METHOD PROTECTED MS_SendingPosition2
VAR_INST
	lrPositionXFirstHalf  	: LREAL;
	lrPositionXSecondHalf  	: LREAL;
	lrPositionYFirstHalf  	: LREAL;
	lrPositionYSecondHalf 	: LREAL;
	lrRotationFirstHalf  	: LREAL;
	lrRotationSecondHalf	: LREAL;
END_VAR
CASE eCR800StateSendPosition OF 
	CR800_SEND_POSITION_CONVERTING:
		LTRUNC( lr_in := lrPositionX2,
				LTRUNC => lrPositionXFirstHalf);
		LTRUNC( lr_in := lrPositionY2,
				LTRUNC => lrPositionYFirstHalf);
		LTRUNC( lr_in := lrRotation2,
				LTRUNC => lrRotationFirstHalf);
	
		FRAC( lr_in := lrPositionX2,
				FRAC => lrPositionXSecondHalf);
		FRAC( lr_in := lrPositionY2,
				FRAC => lrPositionYSecondHalf);
		FRAC( lr_in := lrRotation2,
				FRAC => lrRotationSecondHalf);
				
		eCR800StateSendPosition := CR800_SEND_POSITION_SENDING;
		
	CR800_SEND_POSITION_SENDING:
		stCR800EthercatData.arrRegistersOutput[6028] :=	LREAL_TO_INT(lrPositionXFirstHalf); 
		stCR800EthercatData.arrRegistersOutput[6029] :=	LREAL_TO_INT(1000 * lrPositionXSecondHalf); 
		stCR800EthercatData.arrRegistersOutput[6030] :=	LREAL_TO_INT(lrPositionYFirstHalf); 
		stCR800EthercatData.arrRegistersOutput[6031] :=	LREAL_TO_INT(1000 * lrPositionYSecondHalf); 
		stCR800EthercatData.arrRegistersOutput[6032] :=	LREAL_TO_INT(lrRotationFirstHalf); 
		stCR800EthercatData.arrRegistersOutput[6033] :=	LREAL_TO_INT(1000 * lrRotationSecondHalf); 
			
		eCR800State := CR800_SEND_POSITION_2_DONE;
		
END_CASE
END_METHOD

METHOD PROTECTED MS_SendingPosition2Done
IF NOT bSendPosition2 THEN
	eCR800State := eCR800StateBeforeSendPosition;
	bBusy := FALSE;
	
END_IF
END_METHOD

METHOD Protected MS_Uninitialized
VAR_inst
	iLoop: INT;
END_VAR
//M_ResetVariables();

//M_OperationRigtsEnable(bRequest 	:= 0);
//eCR800StateDoRequest				:= 0 ;
eCR800StateHome 					:= 0 ;	
//eCR800StateReceiveCommand			:= 0 ;
//eCR800SendCommand					:= 0 ;
//eCR800StateInitializing 			:= 0 ;
eCR800StateCycleStop 				:= 0 ; 
eCR800StateCyclePause				:= 0 ; 
eCR800StateSendPosition				:= 0 ;

eErrorID := CR800_ERROR_OK;

bUninitialized := TRUE;
bInit := FALSE;
bGoHome := FALSE;
bUpdateRecipes := FALSE;
bGoAuto := FALSE;
bDoAction := FALSE;
bCycleStop := FALSE;
bCyclePause := FALSE;
bRestoreAuto := FALSE;
bRestoreCycle := FALSE;
bAbort := FALSE;
bError := FALSE;
bAutoModeStarted := FALSE;
bIsHomed := FALSE;
bReset := FALSE;
bStopped := FALSE;
bActive := FALSE; 
	
IF ServoIsOn THEN
	MR_Abort();
END_IF
END_METHOD

METHOD PROTECTED MS_UpdateRecipiesDone
IF NOT bUpdateRecipes THEN
	eCR800State := CR800_IDLE_HOMED ;
END_IF
END_METHOD

METHOD PROTECTED MS_UpdatingRecipies
IF M_DoRequest(iNumberOfRequest := E_RobotSystemActions.UPDATE_RECIPIES) THEN
	eCR800State := CR800_UPDATE_RECIPIES_DONE ;
END_IF
END_METHOD

PROPERTY Name : STRING
GET
Name := sName;
END_GET
SET
sName := Name;
END_SET
END_PROPERTY

(* Desription from CR800 side: Sets the validity of the operation rights for the
external signal control.. *)
{attribute 'monitoring' := 'variable'}
PROPERTY OperationRightsEnable : BOOL
GET
OperationRightsEnable := stCR800EthercatData.arrSignalsOutputConverted[6004] ;
END_GET
SET
stCR800EthercatData.arrSignalsOutputConverted[6004] := OperationRightsEnable ;
END_SET
END_PROPERTY

(*Desription from CR800 side:
Outputs the operation rights valid state for the
external signal control.
The operation right is given when the
operation right input signal is ON, the
controller mode is set to AUTOMATIC, and
there is no other device that currently has the
operation right.*)
{attribute 'monitoring' := 'variable'}
PROPERTY PUBLIC OperationRightsEnabled : BOOL
GET
OperationRightsEnabled := stCR800EthercatData.arrSignalsInputConverted[6004] ;
END_GET
END_PROPERTY

(* Reqest number that robot has to perform *)
{attribute 'monitoring' := 'variable'}
PROPERTY Override : USINT
GET
//Override :=	INT_TO_USINT(stCR800EthercatData.arrRegistersOutput[6021]);
Override := iOverride;
END_GET
SET
//stCR800EthercatData.arrRegistersOutput[6021] := USINT_TO_INT(iOverride);
iOverride := Override;
END_SET
END_PROPERTY

(* Desription from CR800 side:
"This output indicates that the program is
paused.
Turns ON when there is not slot multitask
running, and at least one slot is pausing.
However, slots whose starting condition is set
to ALWAYS or ERROR via a parameter
""SLT**"" will not be executed." *)
{attribute 'monitoring' := 'variable'}
PROPERTY PUBLIC Pausing : BOOL
GET
Pausing := stCR800EthercatData.arrSignalsInputConverted[6006] ;
END_GET
END_PROPERTY

(* Desription from CR800 side:
"This output indicates that a program is being
executed. During multitask operation, this
signal turns ON when at least one task slot is
operating.
However, slots whose starting condition is set
to ALWAYS or ERROR via a parameter ""SLT*""
will not be executed." *)
{attribute 'monitoring' := 'variable'}
PROPERTY PUBLIC ProgramOperating : BOOL
GET
ProgramOperating := stCR800EthercatData.arrSignalsInputConverted[6005] ;
END_GET
END_PROPERTY

(* Desription from CR800 side:
"This input cancels the paused status of the
program and brings the executing line to the
top. Executing a program reset makes it
possible to select a program.
In the multitask mode, the program reset is
applied to all task slots.
However, slots whose starting condition is set
to ALWAYS or ERROR via a parameter
""SLT**"" will not be executed." *)
{attribute 'monitoring' := 'variable'}
PROPERTY ProgramReset : BOOL
GET
ProgramReset := stCR800EthercatData.arrSignalsOutputConverted[6009] ;
END_GET
SET
stCR800EthercatData.arrSignalsOutputConverted[6009] := ProgramReset ;
END_SET
END_PROPERTY

(* "Outputs that in the program selection enabled
state.
Turns ON when program are not running or
pausing.
In multitask operation, this output turns ON
when all task slots are neither operating nor
paused.
However, slots whose starting condition is set
to ALWAYS or ERROR via a parameter
""SLT**"" will not be executed" *)
{attribute 'monitoring' := 'variable'}
PROPERTY PUBLIC ProgramSelectionEnabled : BOOL
GET
ProgramSelectionEnabled := stCR800EthercatData.arrSignalsInputConverted[6009] ;
END_GET
END_PROPERTY

(*Desription from CR800 side:
"This input starts a program. To start a specific
program, select the program using the
program selection signal ""PRGSEL"" and
numerical input ""IODATA,"" and then input the
start signal. Note that when the parameter
""PST"" is enabled, the system reads the
program number from the numerical input
(IODATA) and starts the corresponding
program (i.e., program selection becomes no
longer necessary).
All task slots are executed during multitask
operation.
However, slots whose starting condition is set
to ALWAYS or ERROR via a parameter ""SLT*""
will not be executed." *)
{attribute 'monitoring' := 'variable'}
PROPERTY ProgramStart : BOOL ;
GET
ProgramStart := stCR800EthercatData.arrSignalsOutputConverted[6005] ;
END_GET
SET
stCR800EthercatData.arrSignalsOutputConverted[6005] := ProgramStart ;
END_SET
END_PROPERTY

(* Desription from CR800 side:
This input stops the program being executed.
(The specification is the same as for the STOP
parameter.)
Unlike the STOP parameter, signal numbers
can be changed. *)
{attribute 'monitoring' := 'variable'}
PROPERTY ProgramStop2 : BOOL
GET
ProgramStop2 := stCR800EthercatData.arrSignalsOutputConverted[6007] ;
END_GET
SET
stCR800EthercatData.arrSignalsOutputConverted[6007] := ProgramStop2 ;
END_SET
END_PROPERTY

(* Desription from CR800 side:
"This output indicates that the program is
paused.
(The specification is the same as for the STOP
parameter.)" *)
{attribute 'monitoring' := 'variable'}
PROPERTY PUBLIC ProgramStopped : BOOL
GET
ProgramStopped := bStopped; // stCR800EthercatData.arrSignalsInputConverted[6007] ;
END_GET
END_PROPERTY

(* Reqest number that robot has to perform *)
{attribute 'monitoring' := 'variable'}
PROPERTY RequestNumber : UINT
GET
RequestNumber := iActionNumber;
END_GET
SET
stCR800EthercatData.arrRegistersOutput[6010] :=	UINT_TO_INT(RequestNumber);
END_SET
END_PROPERTY

PROPERTY SendingPosition1 : REFERENCE TO BOOL
GET
SendingPosition1 REF= bSendPosition1;
END_GET
END_PROPERTY

PROPERTY SendingPosition2 : REFERENCE TO BOOL
GET
SendingPosition2 REF= bSendPosition2;
END_GET
END_PROPERTY

(* Desription from a CR800 side:
"This input turns OFF the servo power supply
for the robot.(Applicable to all mechanisms)
The servo cannot be turned ON while this
signal is being input. *)
{attribute 'monitoring' := 'variable'}
PROPERTY PUBLIC ServoIsOff : BOOL
GET
ServoIsOff := NOT ServoIsOn AND CR800PoweredOn; //stCR800EthercatData.arrSignalsInputConverted[6012] ;
END_GET
END_PROPERTY

(* Desription from the CR800 side:
"This output turns ON when the servo power
supply for the robot is ON. If the servo power
supply is OFF, this output also remains OFF.
With a multi-mechanism configuration, this
output turns ON when the servo of at least one
mechanism is ON." *)
{attribute 'monitoring' := 'variable'}
PROPERTY PUBLIC ServoIsOn : BOOL
GET
ServoIsOn := stCR800EthercatData.arrSignalsInputConverted[6011] ;
END_GET
END_PROPERTY

(* Desription from a CR800 side:
"This input turns OFF the servo power supply
for the robot.(Applicable to all mechanisms)
The servo cannot be turned ON while this
signal is being input." *)
{attribute 'monitoring' := 'variable'}
PROPERTY ServoOFF : BOOL
GET
ServoOFF := stCR800EthercatData.arrSignalsOutputConverted[6012] ;
END_GET
SET
stCR800EthercatData.arrSignalsOutputConverted[6012] := ServoOFF ;
END_SET
END_PROPERTY

(* Descrition from the CR800 side:
"This input turns ON the servo power supply for
the robot.
With a multi-mechanism configuration, the
servo power supplies for all mechanisms will
be turned ON." *)
{attribute 'monitoring' := 'variable'}
PROPERTY ServoON : BOOL
GET
ServoON := stCR800EthercatData.arrSignalsOutputConverted[6011] ;
END_GET
SET
stCR800EthercatData.arrSignalsOutputConverted[6011] := ServoON ;
END_SET
END_PROPERTY

(* Actual state of main state machine *)
{attribute 'monitoring' := 'variable'}
PROPERTY State : REFERENCE TO E_CR800State
GET
State REF= eCR800State;
END_GET
END_PROPERTY

METHOD Protected StateMachine
VAR
	MS_CycleStopping_Done: INT;
END_VAR
CASE eCR800State OF
	CR800_UNINITIALIZED:
		MS_Uninitialized();
		
	CR800_INITIALIZING:
		MS_Initializing();
		
	CR800_READY_INITIALIZED:
		MS_ReadyInitialized();

	CR800_IDLE_NOT_HOMED:
		MS_IdleNotHomed();
		
	CR800_GOING_HOME:
		MS_GoingHome();
	
	CR800_GOING_HOME_DONE:
		MS_GoHomeDone();
		
	CR800_IDLE_HOMED:
		MS_IdleHomed();

	CR800_UPDATING_RECIPIES	:
		MS_UpdatingRecipies();
		
	CR800_UPDATE_RECIPIES_DONE:
		MS_UpdateRecipiesDone();
		
	CR800_GOING_AUTO:
		MS_GoingAuto();
		
	CR800_GOING_AUTO_DONE:
		MS_GoAutoDone();
		
	CR800_IDLE_AUTO:
		MS_IdleAuto();
		
	CR800_DOING_ACTION:
		MS_DoingAction();
		
	CR800_DOING_ACTION_DONE:
		MS_DoAction_Done();

	CR800_CYCLE_STOPPING:	
		MS_CycleStopping();
		
	CR800_CYCLE_STOPING_DONE:
		MS_CycleStopDone();
		
	CR800_IDLE_AUTO_PAUSED:
		MS_IdleAutoPaused();
		
	CR800_AUTO_RESTORING:
		MS_RestoringAuto();
	
	CR800_AUTO_RESTORING_DONE:
		MS_RestoreAutoDone();
		
	E_CR800State.CR800_CYCLE_PAUSING:
		MS_CyclePausing();
		
	E_CR800State.CR800_CYCLE_PAUSING_DONE:
		MS_CyclePauseDone();
	
	CR800_IDLE_CYCLE_PAUSED:
		MS_IdleCyclePaused();
	
	CR800_CYCLE_RESTORING:
		MS_RestoringCycle();
	
	CR800_CYCLE_RESTORING_DONE:
		MS_RestoreCycleDone();

	CR800_IN_EXTERNAL_ERROR:
		MS_InExternalError();
		
	CR800_SEND_POSITION_1:
		MS_SendingPosition1();
	
	CR800_SEND_POSITION_1_DONE:
		MS_SendingPosition1Done();	
		
	CR800_SEND_POSITION_2:
		MS_SendingPosition2();
	
	CR800_SEND_POSITION_2_DONE:
		MS_SendingPosition2Done();			
		
	CR800_RESET:
		MS_Reset();
		
	CR800_RESET_DONE:
		MS_ResetDone();
		
	CR800_ABORTING:
		MS_Aborting();
					
END_CASE
END_METHOD

(* Desription from CR800 side:
"Outputs that the stop is being input. (Logical
ADD of all devices.)" *)
{attribute 'monitoring' := 'variable'}
PROPERTY PUBLIC StopSTS : BOOL
GET
StopSTS := stCR800EthercatData.arrSignalsInputConverted[6008] ;
END_GET
END_PROPERTY

PROPERTY Uninitialized : REFERENCE TO BOOL
GET
Uninitialized REF= bUninitialized;
END_GET
END_PROPERTY

(*Desription from CR800 side:
This output indicates that the controller mode
is set to AUTOMATIC.*)
{attribute 'monitoring' := 'variable'}
{attribute 'monitoring' := 'call'}
PROPERTY  UserDefinedArea : ST_CR800UserDefinedArea
GET
UserDefinedArea.bArea1 := stCR800EthercatData.arrSignalsInputConverted[6241];
UserDefinedArea.bArea2 := stCR800EthercatData.arrSignalsInputConverted[6242];
UserDefinedArea.bArea3 := stCR800EthercatData.arrSignalsInputConverted[6243];
UserDefinedArea.bArea4 := stCR800EthercatData.arrSignalsInputConverted[6244];
UserDefinedArea.bArea5 := stCR800EthercatData.arrSignalsInputConverted[6245];
UserDefinedArea.bArea6 := stCR800EthercatData.arrSignalsInputConverted[6246];
UserDefinedArea.bArea7 := stCR800EthercatData.arrSignalsInputConverted[6247];
UserDefinedArea.bArea8 := stCR800EthercatData.arrSignalsInputConverted[6248];
END_GET
END_PROPERTY

PROPERTY UserDefinedArea1 : BOOL
GET
UserDefinedArea1 := stCR800EthercatData.arrSignalsInputConverted[6241];
END_GET
END_PROPERTY

PROPERTY UserDefinedArea2 : BOOL
GET
UserDefinedArea2 := stCR800EthercatData.arrSignalsInputConverted[6242];
END_GET
END_PROPERTY

PROPERTY UserDefinedArea3 : BOOL
GET
UserDefinedArea3 := stCR800EthercatData.arrSignalsInputConverted[6243];
END_GET
END_PROPERTY

PROPERTY UserDefinedArea4 : BOOL
GET
UserDefinedArea4 := stCR800EthercatData.arrSignalsInputConverted[6244];
END_GET
END_PROPERTY

PROPERTY UserDefinedArea5 : BOOL
GET
UserDefinedArea5 := stCR800EthercatData.arrSignalsInputConverted[6245];
END_GET
END_PROPERTY

PROPERTY UserDefinedArea6 : BOOL
GET
UserDefinedArea6 := stCR800EthercatData.arrSignalsInputConverted[6246];
END_GET
END_PROPERTY

PROPERTY UserDefinedArea7 : BOOL
GET
UserDefinedArea7 := stCR800EthercatData.arrSignalsInputConverted[6247];
END_GET
END_PROPERTY

PROPERTY UserDefinedArea8 : BOOL
GET
UserDefinedArea8 := stCR800EthercatData.arrSignalsInputConverted[6248];
END_GET
END_PROPERTY

END_FUNCTION_BLOCK

// ---- POUs/Machine/Module/RTCVision/FB_RTCVision.TcPOU
FUNCTION_BLOCK FB_RTCVision
VAR
	bFirstCycle			: BOOL := TRUE;	(* First cycle bit *)
	
	(* TCPIP params *)
	sName 				: STRING;		(* TCP/IP device name for other utilities *)
	sHost				: T_IPv4Addr;	(*  *)
	sAmsNetID 			: T_AmsNetID;	(*  *)
	iPort				: UINT;			(*  *)
	tTimeout			: TIME;			(*  *)
	
	(* Internal status *) 
	_bActive			: BOOL;			(* TCP/IP device initialized and ready to work *)
	_bBusy				: BOOL;			(* TCP/IP device is currently proccesing *)
	_bError				: BOOL;			(* Error occured while executing *)
	_iErrorID			: UDINT;		(* Error ID*)
	
	_bJobStarted		: BOOL;
	_bJobStopped		: BOOL;
	_eResult_Station1	: E_VisionResult;
	_eResult_Station2	: E_VisionResult;
	
	eCameraState		: E_RTCCameraState;		(* Current state of camera connection *)
	eCameraInitState	: E_RTCCameraInitState;		(* Current state of camera initialization *)
	eCameraMethodState	: E_RTCCameraMethodState;

	(* TCPIP communicate with Vision System - Service side is role as sever *)
	fbTcpClient 		: FB_TcpClient ;
	
	(* Messages buffers *)
	stSendData							: ST_TcpBufferData;		(*  *)
	stReciveData 						: ST_TcpBufferData;		(*  *)

	(* Temporary messeges *)
	sSendMessage 						: STRING;				(*  *)
	sReciveMessage						: STRING(1000);			(*  *)
	arrBufferMessage					: ARRAY[0..10] OF STRING;
	iMessageIndex	 					: INT;	
	sNewLine							: STRING := '$R$L';
	
	(* Rising edge trigger *)
	rtError								: R_TRIG; 					(* Rising edge trigger for function block error *)
	
	(* Status inormation and number *)
	iLastStatusCode						: INT; 
	sLastStatusCode						: STRING;

	(* Internal variables of methods *)
	eSetJobNumber							: E_VisionJob;
	eGetJobNumber							: E_VisionJob;
	eVisionResult							: E_VisionResult;
	
END_VAR

(* First cycle procedure *)
IF bFirstCycle THEN
	bFirstCycle := FALSE;
	
END_IF

_bActive := eCameraState >= RTC_CAMERA_READY;

(* Report errors that occur *)
rtError(CLK:=_bError);

IF rtError.Q THEN 
	fbMachineLogger.MR_AddLogs(FUN_MergeStrings5(sName, ' : Error occured (error ID: ', UDINT_TO_STRING(_iErrorID), ')', ''));

END_IF

(* Execute TCP/IP FB and timers *)
fbTcpClient();

(* Execute state machine *)
StateMachine();

PROPERTY Active  : REFERENCE TO BOOL
GET
Active REF= _bActive;
END_GET
END_PROPERTY

PROPERTY Busy : REFERENCE TO BOOL
GET
Busy REF= _bBusy;
END_GET
END_PROPERTY

PROPERTY CurrentJob : UINT
GET
END_GET
SET
END_SET
END_PROPERTY

PROPERTY Error : REFERENCE TO BOOL
GET
Error REF= _bError;
END_GET
END_PROPERTY

PROPERTY ErrorID : REFERENCE TO UDINT
GET
ErrorID REF= _iErrorID;
END_GET
END_PROPERTY

METHOD GetInfor : BOOL
VAR_INPUT
END_VAR
END_METHOD

PROPERTY JobStarted : BOOL
GET
END_GET
END_PROPERTY

PROPERTY JobStopped : BOOL
GET
END_GET
END_PROPERTY

METHOD MR_Abort : BOOL
VAR_INPUT
END_VAR
IF eCameraState >= RTC_CAMERA_READY THEN
	_bBusy := TRUE;
	MR_Abort := FALSE;
	eCameraState := RTC_CAMERA_ABORTING;
	fbMachineLogger.MR_AddLogs(CONCAT(sName,' : abort requested'));	
	
ELSIF eCameraState = RTC_CAMERA_UNINITIALIZED THEN
	_bBusy := FALSE;
	MR_Abort := TRUE;
	fbMachineLogger.MR_AddLogs(CONCAT(sName,' : abort done'));	
	
END_IF
END_METHOD

METHOD MR_Clear : BOOL
VAR_INPUT
END_VAR
IF eCameraState = RTC_CAMERA_IDLE THEN
	_bBusy := TRUE;
	MR_Clear := FALSE;
	eCameraState := RTC_CAMERA_CLEAR_DATA;
	fbMachineLogger.MR_AddLogs(CONCAT(sName,' : Clear data requested'));	
	
ELSIF eCameraState = RTC_CAMERA_METHOD_DONE THEN
	_bBusy := FALSE;
	MR_Clear := TRUE;
	fbMachineLogger.MR_AddLogs(CONCAT(sName,' : Clear data done'));	

END_IF
END_METHOD

METHOD MR_FirstCycle : BOOL
VAR_INPUT
	sCameraName 			: STRING;		(*  *)
	sClientHost				: T_IPv4Addr;	(*  *)
	sClientAmsNetID 		: T_AmsNetID;	(*  *)
	iClientPort				: UINT;			(*  *)
	tTimeout				: TIME;			(*  *)
	
END_VAR
(* Set fixture name *)
THIS^.sName := sCameraName;

(* Set fixture server initial parameters *)
THIS^.fbTcpClient.MR_FirstCycle(	sName 		:= CONCAT('TCP/IP client of ',sCameraName),
									sHost		:= sClientHost,
									sAmsNetID	:= sClientAmsNetID,
									iPort 		:= iClientPort,
									tTimeout 	:= tTimeout);
END_METHOD

METHOD MR_GetBatchInfor : BOOL
VAR_INPUT
END_VAR
IF eCameraState = RTC_CAMERA_IDLE THEN	
	_bBusy := TRUE;
	MR_GetBatchInfor := FALSE;
	eCameraState := RTC_CAMERA_GET_BATCH_DATA;
	fbMachineLogger.MR_AddLogs(CONCAT(sName,' : get batch data requested'));
	
ELSIF eCameraState = RTC_CAMERA_METHOD_DONE THEN
	_bBusy := FALSE;
	MR_GetBatchInfor := TRUE;
	fbMachineLogger.MR_AddLogs(CONCAT(sName,' : get batch data done'));

END_IF
END_METHOD

METHOD MR_GetResult : BOOL
VAR_INPUT
END_VAR
IF eCameraState = RTC_CAMERA_IDLE THEN	
	_bBusy := TRUE;
	MR_GetResult := FALSE;
	eCameraState := RTC_CAMERA_GET_RESULT;
	fbMachineLogger.MR_AddLogs(CONCAT(sName,' : get result requested'));
	
ELSIF eCameraState = RTC_CAMERA_METHOD_DONE THEN
	_bBusy := FALSE;
	MR_GetResult := TRUE;
	fbMachineLogger.MR_AddLogs(CONCAT(sName,' : get result done'));

END_IF
END_METHOD

METHOD MR_Init : BOOL
VAR_INPUT
END_VAR
IF eCameraState = RTC_CAMERA_UNINITIALIZED THEN
	_bBusy := TRUE;
	MR_Init := FALSE;
	eCameraState := RTC_CAMERA_INITIALIZING;
	fbMachineLogger.MR_AddLogs(CONCAT(sName,' : initializing requested'));	

ELSIF eCameraState >= RTC_CAMERA_READY THEN
	_bBusy := FALSE;
	MR_Init := TRUE;
	fbMachineLogger.MR_AddLogs(CONCAT(sName,' : initializing done'));
	
END_IF
END_METHOD

METHOD MR_Reset : BOOL
VAR_INPUT
END_VAR
END_METHOD

METHOD MR_SetJob : BOOL
VAR_INPUT
	eSetJobNumber 		: E_VisionJob;
END_VAR
IF eCameraState = RTC_CAMERA_IDLE THEN
	THIS^.eSetJobNumber := eSetJobNumber;
	_bBusy := TRUE;
	MR_SetJob := FALSE;
	eCameraState := RTC_CAMERA_SET_JOB;
	fbMachineLogger.MR_AddLogs(FUN_MergeStrings4(sName,' : setting job ',TO_STRING(eSetJobNumber),' requested'));
	
ELSIF eCameraState = RTC_CAMERA_METHOD_DONE THEN
	_bBusy := FALSE;
	MR_SetJob := TRUE;
	fbMachineLogger.MR_AddLogs(FUN_MergeStrings4(sName,' : setting job ',TO_STRING(eSetJobNumber),' done'));

END_IF
END_METHOD

METHOD MR_Start : BOOL
VAR_INPUT
END_VAR
IF eCameraState = RTC_CAMERA_IDLE THEN
	_bBusy := TRUE;
	MR_Start := FALSE;
	eCameraState := RTC_CAMERA_START;
	fbMachineLogger.MR_AddLogs(CONCAT(sName,' : Start job requested'));	
	
ELSIF eCameraState = RTC_CAMERA_METHOD_DONE THEN
	_bBusy := FALSE;
	MR_Start := TRUE;
	fbMachineLogger.MR_AddLogs(CONCAT(sName,' : Start job done'));	

END_IF
END_METHOD

METHOD MR_Stop : BOOL
VAR_INPUT
END_VAR
IF eCameraState = RTC_CAMERA_IDLE THEN	
	_bBusy := TRUE;
	MR_Stop := FALSE;
	eCameraState := RTC_CAMERA_STOP;
	fbMachineLogger.MR_AddLogs(CONCAT(sName,' : stop job requested'));
	
ELSIF eCameraState = RTC_CAMERA_METHOD_DONE THEN
	_bBusy := FALSE;
	MR_Stop := TRUE;
	fbMachineLogger.MR_AddLogs(CONCAT(sName,' : stop job done'));

END_IF
END_METHOD

METHOD MR_StopCycle : BOOL
VAR_INPUT
END_VAR
IF eCameraState = RTC_CAMERA_IDLE THEN	
	_bBusy := TRUE;
	MR_StopCycle := FALSE;
	eCameraState := RTC_CAMERA_STOP_CYCLE;
	fbMachineLogger.MR_AddLogs(CONCAT(sName,' : stop current cycle requested'));
	
ELSIF eCameraState = RTC_CAMERA_METHOD_DONE THEN
	_bBusy := FALSE;
	MR_StopCycle := TRUE;
	fbMachineLogger.MR_AddLogs(CONCAT(sName,' : stop current cycle done'));

END_IF
END_METHOD

METHOD PROTECTED MS_Aborting
fbTcpClient.MR_Abort();

IF NOT fbTcpClient.Active THEN 
	//IF M_ResetParameters() THEN
		eCameraState := RTC_CAMERA_UNINITIALIZED;
		
	//END_IF	
END_IF
END_METHOD

METHOD PROTECTED MS_GetJob : BOOL
VAR_INPUT
END_VAR
CASE eCameraMethodState OF
	RTC_CAMERA_METHOD_SEND_COMMAND:
		MEMSET(ADR(sSendMessage),0,SIZEOF(sSendMessage));
		sSendMessage := CONCAT('GJ','$R$L');
		FUN_StringToTcpBufferData(ADR(sSendMessage),ADR(stSendData));
		
		IF fbTcpClient.MR_AppendToSendBuffer(stSendData) THEN
			eCameraMethodState := RTC_CAMERA_METHOD_RECEIVE_RESPONSE;

		END_IF
		
	RTC_CAMERA_METHOD_RECEIVE_RESPONSE:
		stReciveData := fbTcpClient.NextRecivedMessage;
		
		IF stReciveData.iLength > 0 THEN
			MEMSET(ADR(sReciveMessage),0,SIZEOF(sReciveMessage));
			FUN_TcpBufferDataToString(ADR(sReciveMessage),ADR(stReciveData));

			IF sReciveMessage = 'GJ1' THEN
				THIS^.eGetJobNumber := CASE_RECEIVER_E25_0100812762;				
			END_IF
			
			eCameraMethodState := RTC_CAMERA_METHOD_SEND_COMMAND;
			eCameraState := RTC_CAMERA_METHOD_DONE;	
		END_IF
		
END_CASE
END_METHOD

METHOD PROTECTED MS_Idle
;
END_METHOD

METHOD PROTECTED MS_Initializing
CASE eCameraInitState OF
	
	RTC_INIT_CONNECTION:
		fbTcpClient.MR_Init();
		
		IF fbTcpClient.Active THEN
			eCameraInitState := RTC_INIT_CLEAR_BUFFER;
			
		ELSIF fbTcpClient.Error THEN
			_bError := TRUE;
			_iErrorID := fbTcpClient.ErrorID;
			
		END_IF
	
	RTC_INIT_CLEAR_BUFFER:
		fbTcpClient.MR_ClearAllBuffers();
		eCameraInitState := RTC_INIT_WAIT_FOR_CONFIRMATION;
		
		IF fbTcpClient.Error THEN
			_bError := TRUE;
			_iErrorID := fbTcpClient.ErrorID;
			
		END_IF

	RTC_INIT_WAIT_FOR_CONFIRMATION:
		stReciveData := fbTcpClient.NextRecivedMessage;

		IF stReciveData.iLength > 0 THEN
			MEMSET(ADR(sReciveMessage),0,SIZEOF(sReciveMessage));
			FUN_TcpBufferDataToString(ADR(sReciveMessage),ADR(stReciveData));
	
			IF sReciveMessage = 'User Logged In' THEN
				eCameraInitState := RTC_INIT_DONE;
			
			END_IF
		ELSIF fbTcpClient.Error THEN
			_bError := TRUE;
			_iErrorID := fbTcpClient.ErrorID;
			
		END_IF
		
	RTC_INIT_DONE:
		eCameraInitState := RTC_INIT_CONNECTION;
		eCameraState := RTC_CAMERA_READY;
END_CASE
END_METHOD

METHOD PROTECTED MS_MethodDone
IF NOT _bBusy THEN
	eCameraState := RTC_CAMERA_IDLE;
	
END_IF
END_METHOD

METHOD PROTECTED MS_Ready
eCameraState := RTC_CAMERA_IDLE;
END_METHOD

METHOD PROTECTED MS_Result
CASE eCameraMethodState OF
	RTC_CAMERA_METHOD_SEND_COMMAND:
		MEMSET(ADR(sSendMessage),0,SIZEOF(sSendMessage));
		sSendMessage := CONCAT('Result','$R$L');
		FUN_StringToTcpBufferData(ADR(sSendMessage),ADR(stSendData));
		
		IF fbTcpClient.MR_AppendToSendBuffer(stSendData) THEN
			eCameraMethodState := RTC_CAMERA_METHOD_RECEIVE_RESPONSE;

		END_IF
		
	RTC_CAMERA_METHOD_RECEIVE_RESPONSE:
		stReciveData := fbTcpClient.NextRecivedMessage;
		
		IF stReciveData.iLength > 0 THEN
			MEMSET(ADR(sReciveMessage),0,SIZEOF(sReciveMessage));
			FUN_TcpBufferDataToString(ADR(sReciveMessage),ADR(stReciveData));
			
			IF sReciveMessage = 'ResultGood' THEN
				eVisionResult := VISION_RESULT_GOOD;
				
			ELSIF sReciveMessage = 'ResultDirt' THEN
				eVisionResult := VISION_RESULT_CONTAMINATION_DIRTY;
				
			ELSIF sReciveMessage = 'ResultDent' THEN
				eVisionResult := VISION_RESULT_SCRATCH_DENT;
				
			ELSIF sReciveMessage = 'ResultReject' THEN
				eVisionResult := VISION_RESULT_REJECT;
				
			ELSE
				eVisionResult := VISION_RESULT_UNKNOWN;
				
			END_IF			
			eCameraMethodState := RTC_CAMERA_METHOD_SEND_COMMAND;
			eCameraState := RTC_CAMERA_METHOD_DONE;	
			
		END_IF		
END_CASE
END_METHOD

METHOD PROTECTED MS_SetJob
CASE eCameraMethodState OF
	RTC_CAMERA_METHOD_SEND_COMMAND:
		MEMSET(ADR(sSendMessage),0,SIZEOF(sSendMessage));
		sSendMessage := FUN_MergeStrings3('SJ', TO_STRING(TO_INT(THIS^.eSetJobNumber)), '$R$L');
		FUN_StringToTcpBufferData(ADR(sSendMessage),ADR(stSendData));
		
		IF fbTcpClient.MR_AppendToSendBuffer(stSendData) THEN
			eCameraMethodState := RTC_CAMERA_METHOD_RECEIVE_RESPONSE;

		END_IF
		
	RTC_CAMERA_METHOD_RECEIVE_RESPONSE:
		stReciveData := fbTcpClient.NextRecivedMessage;
		
		IF stReciveData.iLength > 0 THEN
			MEMSET(ADR(sReciveMessage),0,SIZEOF(sReciveMessage));
			FUN_TcpBufferDataToString(ADR(sReciveMessage),ADR(stReciveData));
			
			IF sReciveMessage = 'SJDone' THEN
				eCameraMethodState := RTC_CAMERA_METHOD_SEND_COMMAND;
				eCameraState := RTC_CAMERA_METHOD_DONE;			
			END_IF	
		END_IF
		
END_CASE
END_METHOD

METHOD PROTECTED MS_Start
CASE eCameraMethodState OF
	
	RTC_CAMERA_METHOD_SEND_COMMAND:
		MEMSET(ADR(sSendMessage),0,SIZEOF(sSendMessage));
		sSendMessage := CONCAT('Start', '$R$L');
		FUN_StringToTcpBufferData(ADR(sSendMessage),ADR(stSendData));
		
		IF fbTcpClient.MR_AppendToSendBuffer(stSendData) THEN
			eCameraMethodState := RTC_CAMERA_METHOD_RECEIVE_RESPONSE;
							
		END_IF
		
	RTC_CAMERA_METHOD_RECEIVE_RESPONSE:
		stReciveData := fbTcpClient.NextRecivedMessage;
		
		IF stReciveData.iLength > 0 THEN
			MEMSET(ADR(sReciveMessage),0,SIZEOF(sReciveMessage));
			FUN_TcpBufferDataToString(ADR(sReciveMessage),ADR(stReciveData));
			
			IF sReciveMessage = 'StartDone' THEN
				eCameraMethodState := RTC_CAMERA_METHOD_SEND_COMMAND;
				eCameraState := RTC_CAMERA_METHOD_DONE;			
			END_IF	
		END_IF

END_CASE
END_METHOD

METHOD PROTECTED MS_Stop : BOOL
VAR_INPUT
END_VAR
CASE eCameraMethodState OF
	RTC_CAMERA_METHOD_SEND_COMMAND:
		MEMSET(ADR(sSendMessage),0,SIZEOF(sSendMessage));
		sSendMessage := CONCAT('Stop','$R$L');
		FUN_StringToTcpBufferData(ADR(sSendMessage),ADR(stSendData));
		
		IF fbTcpClient.MR_AppendToSendBuffer(stSendData) THEN
			eCameraMethodState := RTC_CAMERA_METHOD_RECEIVE_RESPONSE;

		END_IF
		
	RTC_CAMERA_METHOD_RECEIVE_RESPONSE:
		stReciveData := fbTcpClient.NextRecivedMessage;
		
		IF stReciveData.iLength > 0 THEN
			MEMSET(ADR(sReciveMessage),0,SIZEOF(sReciveMessage));
			FUN_TcpBufferDataToString(ADR(sReciveMessage),ADR(stReciveData));
			
			IF sReciveMessage = 'StopDone' THEN
				eCameraMethodState := RTC_CAMERA_METHOD_SEND_COMMAND;
				eCameraState := RTC_CAMERA_METHOD_DONE;			
			END_IF	
		END_IF
		
END_CASE
END_METHOD

METHOD PROTECTED MS_Uninitialized
;
END_METHOD

METHOD PROTECTED StateMachine : BOOL
VAR_INPUT
END_VAR
CASE eCameraState OF
	RTC_CAMERA_UNINITIALIZED:
		MS_Uninitialized();
	
	RTC_CAMERA_INITIALIZING:
		MS_Initializing();
		
	RTC_CAMERA_READY:
		MS_Ready();
		
	RTC_CAMERA_IDLE:
		MS_Idle();
		
	RTC_CAMERA_SET_JOB:
		MS_SetJob();
		

	
	RTC_CAMERA_METHOD_DONE:
		MS_MethodDone();
		
	RTC_CAMERA_ABORTING:
		MS_Aborting();
END_CASE
END_METHOD

END_FUNCTION_BLOCK

// ---- POUs/Libs/Bowl Feeder/FB_BowlFeeder.TcPOU
(*
Copyrights	: Operation Automation Department
Author		: HVAP
Description	: This function block is used to control bowl feeder REOVIB MFS 268
*)
FUNCTION_BLOCK FB_BowlFeeder IMPLEMENTS I_BowlFeeder
VAR CONSTANT
	(* STRINGS *)
	sPRODUCT_PRESENCE_SENSOR_NAME	: STRING := 'Producr presence sensor';
	sSTATUS_RELAY					: STRING := 'Status relay from bowl driver';
	sENABLE							: STRING := 'Enable bowl driver';
END_VAR
VAR
	bFirstCycle			: BOOL := TRUE;		(* First cycle bit *)
	sName 				: STRING;			(* Bowl Feeder name for other utilities *)	
	
	(* Internal status *)
	_bActive : BOOL;
	_bBusy : BOOL;
	_bError : BOOL;
	_uiErrorID : UINT;
	
	(* State machine *)
	eBowlFeederUnitState 		: E_BowlFeederUnitState;
	eBowlFeederUnitStateInit 	: E_BowlFeederUnitStateInit;
	
	(* Hardware module *)
	//_diProductPresence	: FB_DigitalInput;	(* Sensor for monitoring the queue of components on the track or an input for switching to the second setpoint 24 VDC (PNP). *)
	diStatusRelay		: FB_DigitalInput;	(* Relay closes when the feeder is running – the relay opens when there is no enable signal or a fault displayed. *)
	doEnable			: FB_DigitalOutput;	(* External control function to switch the power output ON or OFF *)
	_aoSetpoint			: FB_AnalogOutput;	(* 0-100%*)
	
	(* Rising edge trigger *)
	rtError								: R_TRIG; 					(* Rising edge trigger for function block error *)
END_VAR
(*
Version history:

+-------------+------------+----------------+----------+------------------------------------------+
|Date         | Version    | created under  | Author   | Remark                                   |
+=============+============+================+==========+==========================================+
|2024-02      | 1.0.0.0    | V3.1.4024.22   | HVAP     | Function block created                   |
+-------------+------------+----------------+----------+------------------------------------------+

*)

IF bFirstCycle THEN
	bFirstCycle := FALSE;
	
//	_diProductPresence.MR_FirstCycle( 	sName 		:= CONCAT(STR1:= sName, STR2:= CONCAT(STR1:= ':', STR2:= sPRODUCT_PRESENCE_SENSOR_NAME)),
//										sModuleType := '',
//										sPortID 	:= '');
	
	diStatusRelay.MR_FirstCycle(	sName		:= CONCAT(STR1:= sName, STR2:= CONCAT(STR1:= ':', STR2:= sSTATUS_RELAY)),
									sModuleType	:= '',
									sPortID		:= '');
									
	doEnable.MR_FirstCycle(	sName		:= CONCAT(STR1:= sName, STR2:= CONCAT(STR1:= ':', STR2:= sENABLE)),
							sModuleType	:= '',
							sPortID		:= '');
END_IF

(* Ready to work *)
_bActive := eBowlFeederUnitState >= BOWL_FEEDER_UNIT_IDLE;
_bBusy := eBowlFeederUnitState <> BOWL_FEEDER_UNIT_IDLE AND eBowlFeederUnitState <> BOWL_FEEDER_UNIT_UNINITIALIZED;

(* Report errors that occur *)
rtError(CLK:=_bError);
IF rtError.Q THEN 
	fbMachineLogger.MR_AddLogs(CONCAT(sName, ' : Error occured'));
END_IF

StateMachine();

PROPERTY Active : BOOL
GET
Active := _bActive;
END_GET
END_PROPERTY

PROPERTY Busy : BOOL
GET
Busy := _bBusy;
END_GET
END_PROPERTY

PROPERTY Error : BOOL
GET
Error := _bError;
END_GET
END_PROPERTY

PROPERTY ErrorID : UINT
GET
ErrorID := _uiErrorID;
END_GET
END_PROPERTY

METHOD MR_FirstCycle : BOOL
VAR_INPUT
	sName	: STRING;
END_VAR
THIS^.sName := sName;
END_METHOD

METHOD MR_Init : BOOL
VAR_INPUT
END_VAR
IF eBowlFeederUnitState = BOWL_FEEDER_UNIT_UNINITIALIZED THEN
	MR_Init := FALSE;
	eBowlFeederUnitState := BOWL_FEEDER_UNIT_INITIALIZING;	
	fbMachineLogger.MR_AddLogs(CONCAT(sName,': initializing requested'));
		
ELSIF eBowlFeederUnitState >= BOWL_FEEDER_UNIT_READY_INITIALIZED THEN
	MR_Init := TRUE;
	fbMachineLogger.MR_AddLogs(CONCAT(sName,': initializing done'));

END_IF
END_METHOD

METHOD MR_Start : BOOL
VAR_INPUT
END_VAR
IF eBowlFeederUnitState = BOWL_FEEDER_UNIT_IDLE THEN
	MR_Start := FALSE;
	eBowlFeederUnitState := BOWL_FEEDER_UNIT_START;
	fbMachineLogger.MR_AddLogs(CONCAT(sName,': Start requesting'));
		
ELSIF eBowlFeederUnitState = BOWL_FEEDER_UNIT_RUNNING THEN
	MR_Start := TRUE;
	fbMachineLogger.MR_AddLogs(CONCAT(sName,': Start done, is running'));
	
END_IF
END_METHOD

METHOD MR_Stop : BOOL
VAR_INPUT
END_VAR
IF eBowlFeederUnitState = BOWL_FEEDER_UNIT_IDLE THEN
	MR_Stop := FALSE;
	eBowlFeederUnitState := BOWL_FEEDER_UNIT_STOP;
	fbMachineLogger.MR_AddLogs(CONCAT(sName,': Stop requesting'));

ELSIF eBowlFeederUnitState = BOWL_FEEDER_UNIT_IDLE THEN
	MR_Stop := TRUE;
	fbMachineLogger.MR_AddLogs(CONCAT(sName,': Stop done'));
	
END_IF
END_METHOD

METHOD MS_Abort
doEnable.Out := FALSE;

IF NOT diStatusRelay.In THEN
	(* Status bit *)
	_bError		:= FALSE;
	
	(* State transition *)
	eBowlFeederUnitState := BOWL_FEEDER_UNIT_UNINITIALIZED;
END_IF
END_METHOD

METHOD PROTECTED MS_Idle
;
END_METHOD

METHOD PROTECTED MS_Initializing
CASE eBowlFeederUnitStateInit OF
	BOWL_FEEDER_UNIT_INIT_START:
		doEnable.Out := TRUE;
		eBowlFeederUnitStateInit := BOWL_FEEDER_UNIT_INIT_RUNNING_CHECK;
		
	BOWL_FEEDER_UNIT_INIT_RUNNING_CHECK:
		IF diStatusRelay.In THEN
			eBowlFeederUnitStateInit := BOWL_FEEDER_UNIT_INIT_STOP;
		END_IF
	
	BOWL_FEEDER_UNIT_INIT_STOP:
		doEnable.Out := FALSE;
		eBowlFeederUnitStateInit := BOWL_FEEDER_UNIT_INIT_STOP_CHECK;
		
	BOWL_FEEDER_UNIT_INIT_STOP_CHECK:
		IF NOT diStatusRelay.In THEN
			eBowlFeederUnitStateInit := BOWL_FEEDER_UNIT_INIT_DONE;
		END_IF
		
	BOWL_FEEDER_UNIT_INIT_DONE:
		eBowlFeederUnitStateInit := BOWL_FEEDER_UNIT_INIT_START;
		eBowlFeederUnitState := BOWL_FEEDER_UNIT_READY_INITIALIZED;
		
END_CASE
END_METHOD

METHOD PROTECTED MS_Ready
eBowlFeederUnitState := BOWL_FEEDER_UNIT_IDLE;
END_METHOD

METHOD MS_Running
eBowlFeederUnitState := BOWL_FEEDER_UNIT_IDLE;
END_METHOD

METHOD PROTECTED MS_Start : BOOL
VAR_INPUT
END_VAR
doEnable.Out := TRUE;

IF diStatusRelay.In THEN
	eBowlFeederUnitState := BOWL_FEEDER_UNIT_RUNNING;
END_IF
END_METHOD

METHOD MS_Stop
doEnable.Out := FALSE;

IF NOT diStatusRelay.In THEN
	eBowlFeederUnitState := BOWL_FEEDER_UNIT_STOP_DONE;
END_IF
END_METHOD

METHOD MS_StopDone
eBowlFeederUnitState := BOWL_FEEDER_UNIT_IDLE;
END_METHOD

METHOD PROTECTED MS_Uninitialized
;
END_METHOD

PROPERTY Running : BOOL
GET
Running := diStatusRelay.In;
END_GET
END_PROPERTY

PROPERTY Setpoint : REAL
GET
Setpoint := _aoSetpoint.Value;
END_GET
SET
_aoSetpoint.Value := Setpoint;
END_SET
END_PROPERTY

METHOD PROTECTED StateMachine
CASE eBowlFeederUnitState OF
	BOWL_FEEDER_UNIT_UNINITIALIZED:
		MS_Uninitialized();
		
	BOWL_FEEDER_UNIT_INITIALIZING:
		MS_Initializing();
		
	BOWL_FEEDER_UNIT_READY_INITIALIZED:
		MS_Ready();
		
	BOWL_FEEDER_UNIT_IDLE:
		MS_Idle();
		
	BOWL_FEEDER_UNIT_START:
		MS_Start();
		
	BOWL_FEEDER_UNIT_RUNNING:
		MS_Running();
		
	BOWL_FEEDER_UNIT_STOP:
		MS_Stop();
		
	BOWL_FEEDER_UNIT_STOP_DONE:
		MS_StopDone();
		
	BOWL_FEEDER_UNIT_ABORT:
		MS_Abort();
	
END_CASE
END_METHOD

END_FUNCTION_BLOCK

// ---- POUs/Libs/Analog Devices/Analog Output/FB_AnalogOutput.TcPOU
(* 
| :Description: This function block represents basic analog output and can be used for creating an instance of analog output device. 
| To control the output state use property "Out" 
*)
FUNCTION_BLOCK FB_AnalogOutput EXTENDS FB_AnalogDevice IMPLEMENTS I_AnalogOutput
VAR
	intAnalogOut AT %Q* : INT; (* Analog output value 0-32767 *)
	rConvertedValue : REAL;
END_VAR
(*
Version history:

+-------------+------------+----------------+----------+------------------------------------------+
|Date         | Version    | created under  | Author   | Remark                                   |
+=============+============+================+==========+==========================================+
|2024-02      | 1.0.0.0    | V3.1.4024.22   | HVAP     | Function block created                   |
+-------------+------------+----------------+----------+------------------------------------------+

*)

(*
Analog output
0-10V : 0-32767 : 0-100%
*)

PROPERTY Value : REAL
GET
Value := (INT_TO_REAL(intAnalogOut)/32767.0)*100.0;
END_GET
SET
intAnalogOut := REAL_TO_INT((Value/(100.0 - 0.0))*(32767.0 - 0.0));
END_SET
END_PROPERTY

END_FUNCTION_BLOCK

// ---- POUs/Libs/Analog Devices/Analog Device/FB_AnalogDevice.TcPOU
(* 
:Description: This function block is base for all other analog devices.
*)
FUNCTION_BLOCK ABSTRACT FB_AnalogDevice IMPLEMENTS I_AnalogDevice
VAR
	sName 		: STRING; (* Name of analog device instance *)
	sModuleType : STRING; (* Name of analog device instance *)
	sPortID		: STRING; (* Slot number on the module *)
END_VAR
(*
Version history:

+-------------+------------+----------------+----------+------------------------------------------+
|Date         | Version    | created under  | Author   | Remark                                   |
+=============+============+================+==========+==========================================+
|2024-02      | 1.0.0.0    | V3.1.4024.22   | HVAP     | Function block created                   |
+-------------+------------+----------------+----------+------------------------------------------+

*)

PROPERTY ModuleType : REFERENCE TO STRING
GET
ModuleType REF= sModuleType;
END_GET
END_PROPERTY

(*
:Description: Call this method in the first cycle of the program
*)
METHOD MR_FirstCycle : BOOL
VAR_INPUT
	sName		: STRING;
	sModuleType	: STRING;
	sPortID		: STRING;
END_VAR
THIS^.sName 		:= sName;
THIS^.sModuleType 	:= sModuleType;
THIS^.sPortID 		:= sPortID;
END_METHOD

PROPERTY Name : REFERENCE TO STRING
GET
Name REF= sName;
END_GET
END_PROPERTY

PROPERTY PortID : REFERENCE TO STRING
GET
PortID REF= sPortID;
END_GET
END_PROPERTY

END_FUNCTION_BLOCK

// ---- POUs/Machine/Module/RTCVision/FB_DoubleTrigger.TcPOU
FUNCTION_BLOCK FB_DoubleTrigger
VAR
	doCam : FB_DigitalOutput;
END_VAR

METHOD Command : BOOL
VAR_INPUT	
	PulseWidth	: TIME; //T#0.1ms
	DelayTimeForSecondTrigger	: TIME; //T#0.1ms
END_VAR
VAR_INST
	uiState 					: UINT;
	tonDelay					: TON;
END_VAR
CASE uiState OF
	0://first trigger on
		doCam.Out := TRUE;
		uiState := 10;
	10://first trigger off
		tonDelay(IN := TRUE, PT := PulseWidth);
		IF tonDelay.Q THEN	
			doCam.Out := FALSE;	
			tonDelay(IN := FALSE);
			uiState := 20;
		END_IF
	20://second trigger on
		tonDelay(IN := TRUE, PT := DelayTimeForSecondTrigger);
		IF tonDelay.Q THEN	
			doCam.Out := TRUE;
			tonDelay(IN := FALSE);
			uiState := 30;
		END_IF
	30://second trigger off
		tonDelay(IN := TRUE, PT := PulseWidth); 
		IF tonDelay.Q THEN
			doCam.Out := FALSE;
			tonDelay(IN := FALSE);
			Command := TRUE;
			uiState := 0;
		END_IF
END_CASE
END_METHOD

END_FUNCTION_BLOCK

// ---- POUs/Libs/Utilities/FB_DataSetFifo_1.TcPOU
FUNCTION_BLOCK FB_DataSetFifo_1
VAR_INPUT
	bOverwrite	: BOOL;
	in 			: LREAL;
END_VAR
VAR_OUTPUT
	bOk			: BOOL;
	nCount		: UDINT;
	nLoad		: UDINT;
	out			: LREAL;
END_VAR
VAR
	arrBuffer 	: ARRAY[0..10000] OF BYTE; (* Buffer memory used by FB_MemRingBuffer function block *)
	fbBuffer	: FB_MemRingBuffer;
END_VAR

;

ACTION A_Add:
fbBuffer.A_AddTail( pWrite:= ADR( in ),
					cbWrite:= SIZEOF( in ),
					pBuffer:= ADR( arrBuffer ),
					cbBuffer:= SIZEOF( arrBuffer ),
					bOk=> bOk,
					nCount => nCount );


IF NOT bOk THEN (* overflow ? *)
	IF bOverwrite THEN
		fbBuffer.A_RemoveHead(); (* remove one oldest entry *)

		fbBuffer.A_AddTail( bOk => bOk, nCount => nCount );
	END_IF
END_IF



nLoad := (fbBuffer.cbSize * 100) / 10000;
END_ACTION

ACTION A_Get:
fbBuffer.A_GetHead( pRead:= ADR( out ),
					cbRead:= SIZEOF( out ),
					pBuffer:= ADR( arrBuffer ),
					cbBuffer:= SIZEOF( arrBuffer ),
					bOk=> bOk,
					nCount => nCount );

nLoad := (fbBuffer.cbSize * 100) / 10000;
END_ACTION

ACTION A_Remove:
fbBuffer.A_RemoveHead( 	pRead:= ADR( out ),
						cbRead:= SIZEOF( out ),
						pBuffer:= ADR( arrBuffer ),
						cbBuffer:= SIZEOF( arrBuffer ),
						bOk=> bOk,
						nCount => nCount );

nLoad := (fbBuffer.cbSize * 100) / 10000;
END_ACTION

ACTION A_Reset:
MEMSET( ADR( arrBuffer ), 0, SIZEOF( arrBuffer ) ); (* reset (optional) internal buffer *)

fbBuffer.A_Reset( 	bOk=> bOk,
					nCount => nCount );

nLoad := (fbBuffer.cbSize * 100) / 10000;
END_ACTION

END_FUNCTION_BLOCK

// ---- POUs/Libs/Utilities/FB_DataSetFifo.TcPOU
FUNCTION_BLOCK FB_DataSetFifo
VAR
	arrBuffer 	: ARRAY[0..10000] OF BYTE; (* Buffer memory used by FB_MemRingBuffer function block *)
	fbBuffer	: FB_MemRingBuffer;
	
	_bOk		: BOOL;
	_nCount		: UDINT;
	_nLoad		: UDINT;
	_bOverwrite	: BOOL;
END_VAR

METHOD Add1Data : BOOL
VAR_INPUT
	in : LREAL;
END_VAR
fbBuffer.A_AddTail( pWrite:= ADR( in ),
					cbWrite:= SIZEOF( in ),
					pBuffer:= ADR( arrBuffer ),
					cbBuffer:= SIZEOF( arrBuffer ),
					bOk=> _bOk,
					nCount => _nCount );

Add1Data := _bOk;
//IF NOT _bOk THEN (* overflow ? *)
//	IF bOverwrite THEN
//		fbBuffer.A_RemoveHead(); (* remove one oldest entry *)

//		fbBuffer.A_AddTail( bOk => _bOk, nCount => _nCount );
//	END_IF
//END_IF



_nLoad := (fbBuffer.cbSize * 100) / 1000;
END_METHOD

METHOD Add2Data : BOOL
VAR_INPUT
	in1 : LREAL;
	in2	: LREAL;
END_VAR
VAR_INST
	Add2DataStep : UINT;
	bOktemp			: BOOL;
END_VAR
CASE Add2DataStep OF
	0:
		fbBuffer.A_AddTail( pWrite:= ADR( in1 ),
					cbWrite:= SIZEOF( in1 ),
					pBuffer:= ADR( arrBuffer ),
					cbBuffer:= SIZEOF( arrBuffer ),
					bOk=> bOktemp,
					nCount => _nCount );
		IF bOktemp THEN
			fbBuffer.A_AddTail( pWrite:= ADR( in2 ),
					cbWrite:= SIZEOF( in2 ),
					pBuffer:= ADR( arrBuffer ),
					cbBuffer:= SIZEOF( arrBuffer ),
					bOk=> _bOk,
					nCount => _nCount );
			IF _bOk THEN
				Add2DataStep := 1;
			END_IF
		END_IF
	1: //done
		_nLoad := (fbBuffer.cbSize * 100) / 1000;
		Add2Data := TRUE;
		Add2DataStep := 0;
END_CASE
END_METHOD

PROPERTY Count : REFERENCE TO UDINT
GET
Count REF= _nCount;
END_GET
END_PROPERTY

METHOD GetData : BOOL
VAR_OUTPUT
	out : LREAL;
END_VAR
fbBuffer.A_GetHead( pRead:= ADR( out ),
					cbRead:= SIZEOF( out ),
					pBuffer:= ADR( arrBuffer ),
					cbBuffer:= SIZEOF( arrBuffer ),
					bOk=> _bOk,
					nCount => _nCount );
GetData := _bOk;
_nLoad := (fbBuffer.cbSize * 100) / 1000;
END_METHOD

PROPERTY GetValue : LREAL (*Auto remove value after get *)
GET
(*
Description: Get the first value in the buffer, not remove it.
*)
VAR
END_VAR
fbBuffer.A_GetHead( 	pRead:= ADR( GetValue ),
						cbRead:= SIZEOF( GetValue ),
						pBuffer:= ADR( arrBuffer ),
						cbBuffer:= SIZEOF( arrBuffer ),
						bOk=> _bOk,
						nCount => _nCount );

_nLoad := (fbBuffer.cbSize * 100) / 1000;
END_GET
END_PROPERTY

PROPERTY Load : UDINT
GET
Load := _nLoad;
END_GET
END_PROPERTY

PROPERTY OK : REFERENCE TO BOOL
GET
OK REF= _bOk;
END_GET
END_PROPERTY

PROPERTY OverWrite : BOOL
SET
_bOverwrite := OverWrite;
END_SET
END_PROPERTY

METHOD Remove : BOOL
VAR_OUTPUT
	out : LREAL;
END_VAR
fbBuffer.A_RemoveHead( 	pRead:= ADR( out ),
						cbRead:= SIZEOF( out ),
						pBuffer:= ADR( arrBuffer ),
						cbBuffer:= SIZEOF( arrBuffer ),
						bOk=> _bOk,
						nCount => _nCount );
Remove := _bOk;
_nLoad := (fbBuffer.cbSize * 100) / 1000;
END_METHOD

METHOD Reset : BOOL
VAR_INPUT
END_VAR
MEMSET( ADR( arrBuffer ), 0, SIZEOF( arrBuffer ) ); (* reset (optional) internal buffer *)

fbBuffer.A_Reset( 	bOk=> _bOk,
					nCount => _nCount );

_nLoad := (fbBuffer.cbSize * 100) / 1000;
END_METHOD

END_FUNCTION_BLOCK

// ---- POUs/Libs/Alarms/VisuEvents/FB_VisuEventsHandling.TcPOU
FUNCTION_BLOCK ABSTRACT FB_VisuEventsHandling EXTENDS FB_ListenerBase
VAR
	arrEvents				: ARRAY[1..iMAX_EVENTS] OF ST_Event;		//Dla HMI (*  *)
	arrActiveAlarms			: ARRAY[1..iMAX_EVENTS] OF ST_Event;		//Dla HMI (*  *)
	arrActiveEvents			: ARRAY[1..iMAX_DEFINITION_EVENTS] OF ST_BaseEvent;	(*  *)
	
	iActiveDefinitionEvents	: UDINT;	(* the contents of the arrActiveEvents table *)
	iActiveAlarms			: UDINT;	(* the contents of the alarm table *)
	
	iActiveCritical			: UDINT;	(*  *)
	iActiveError			: UDINT;	(*  *)
	iActiveWarning			: UDINT;	(*  *)
	iActiveInfo				: UDINT;	(*  *)
	iActiveVerbose			: UDINT;	(*  *)
	
	bSummertime				: BOOL;		(*  *)
END_VAR

Execute();

METHOD Execute : HRESULT
VAR_INPUT
END_VAR
VAR_INST
	fbRequestEventText  : FB_RequestEventText;
	stBaseEvent 		: ST_BaseEvent;
	bReqText 			: BOOL;
	{attribute 'TcEncoding':='UTF-8'}
	sLastMessageText 	: STRING;
	index				: udint;
END_VAR
VAR
	rtAlarmCleard : R_TRIG;
END_VAR
Execute := SUPER^.Execute(); //retrieve events

IF iActiveDefinitionEvents > 0 AND bReqText = FALSE THEN
	stBaseEvent := arrActiveEvents[iActiveDefinitionEvents];
	fbRequestEventText.Request(eventClass:=stBaseEvent.guidEventClass, nEventId:=stBaseEvent.iEventId, nLangId := Tc3_EventLogger.GVL.nLangId_OnlineMonitoring, ipArgs:=stBaseEvent.iTcArguments);
	MEMSET(ADR(arrActiveEvents[iActiveDefinitionEvents]),0,SIZEOF(arrActiveEvents[iActiveDefinitionEvents]));
	iActiveDefinitionEvents := iActiveDefinitionEvents - 1;
	bReqText := TRUE;
END_IF

//retrieve the text of a message
IF 	bReqText AND fbRequestEventText.bError THEN 
	sLastMessageText := 'Error';
	bReqText := FALSE;
ELSIF bReqText AND NOT fbRequestEventText.bBusy THEN
	rtAlarmCleard(CLK := stBaseEvent.eEventType = E_EventType.ALARM_CLEARED); //RMA
	IF stBaseEvent.eEventType = E_EventType.MESSAGE OR stBaseEvent.eEventType = E_EventType.ALARM_RAISED THEN
		MEMCPY(ADR(arrEvents[2]),ADR(arrEvents[1]),SIZEOF(arrEvents[1]) * (iMAX_EVENTS - 1));
		fbRequestEventText.GetString(sLastMessageText, SIZEOF(sLastMessageText));
		arrEvents[1].iType := stBaseEvent.iType;
		arrEvents[1].eSeverity := stBaseEvent.eSeverity;
		arrEvents[1].iEventId := stBaseEvent.iEventId;
		arrEvents[1].guidEventClass := stBaseEvent.guidEventClass;
		arrEvents[1].sSourceName := stBaseEvent.sSourceName;
		arrEvents[1].iSourceID := stBaseEvent.iSourceID;
		//arrEvents[1].nTimeStamp := ULINT_TO_DT(stBaseEvent.nTimeStamp/10000000 - 11644473600); //100ns -> s - 1601.01.01:00:00:00
		arrEvents[1].iTimeStamp := stBaseEvent.iTimeStamp/10000 - 11644473600000; //100ns to ms -> /1000
		arrEvents[1].iTimeStampCleared := 0; //100ns to ms -> /1000
		arrEvents[1].iTimeStampConfirmed :=0; //100ns to ms -> /1000
		IF NOT bSummertime THEN
			arrEvents[1].iTimeStamp := arrEvents[1].iTimeStamp + 3600000;
		END_IF
		UTF8_TO_STRING(pDstSTRING:=ADR(arrEvents[1].sEventText), pSrcUTF8:=ADR(sLastMessageText), nDstSize:=SIZEOF(arrEvents[1].sEventText), nDstLen=> );
		IF LEN2(ADR(stBaseEvent.sJsonAttribute)) > 0 THEN
			//arrEvents[1].wsJsonAttribute := stBaseEvent.wsJsonAttribute;
			FindAndReplaceChar(
				pSrcString:= ADR(stBaseEvent.sJsonAttribute), 
				sDeleteChar:= '"', 
				sInsertChar:= '', 
				pDstString:= ADR(arrEvents[1].sJsonAttribute), 
				nDstSize:= LEN2(ADR(stBaseEvent.sJsonAttribute)));
			FindAndReplaceChar(
				pSrcString:= ADR(arrEvents[1].sJsonAttribute), 
				sDeleteChar:= ':', 
				sInsertChar:= '$T', 
				pDstString:= ADR(arrEvents[1].sJsonAttribute), 
				nDstSize:= LEN2(ADR(arrEvents[1].sJsonAttribute)));
			FindAndReplaceChar(
				pSrcString:= ADR(arrEvents[1].sJsonAttribute), 
				sDeleteChar:= ',', 
				sInsertChar:= '$N', 
				pDstString:= ADR(arrEvents[1].sJsonAttribute), 
				nDstSize:= LEN2(ADR(arrEvents[1].sJsonAttribute)));
			FindAndReplaceChar(
				pSrcString:= ADR(arrEvents[1].sJsonAttribute), 
				sDeleteChar:= '{', 
				sInsertChar:= '', 
				pDstString:= ADR(arrEvents[1].sJsonAttribute), 
				nDstSize:= LEN2(ADR(arrEvents[1].sJsonAttribute)));
			FindAndReplaceChar(
				pSrcString:= ADR(arrEvents[1].sJsonAttribute), 
				sDeleteChar:= '}', 
				sInsertChar:= '', 
				pDstString:= ADR(arrEvents[1].sJsonAttribute), 
				nDstSize:= LEN2(ADR(arrEvents[1].sJsonAttribute)));							
		END_IF	
		arrEvents[1].sEventText := arrEvents[1].sEventText;
		//aktywne alarmy
		IF stBaseEvent.eEventType = E_EventType.ALARM_RAISED THEN
			MEMCPY(ADR(arrActiveAlarms[2]),ADR(arrActiveAlarms[1]),SIZEOF(arrActiveAlarms[1]) * (iMAX_EVENTS - 1));
			arrActiveAlarms[1].iType 			:= arrEvents[1].iType;
			arrActiveAlarms[1].eSeverity 		:= arrEvents[1].eSeverity;
			arrActiveAlarms[1].iEventId 		:= arrEvents[1].iEventId;
			arrActiveAlarms[1].iTimeStamp 		:= arrEvents[1].iTimeStamp;
			arrActiveAlarms[1].sEventText 		:= arrEvents[1].sEventText;
			arrActiveAlarms[1].sJsonAttribute 	:= arrEvents[1].sJsonAttribute;
			arrActiveAlarms[1].guidEventClass 	:= arrEvents[1].guidEventClass;
			arrActiveAlarms[1].sSourceName 		:= arrEvents[1].sSourceName;
			arrActiveAlarms[1].iSourceID 		:= arrEvents[1].iSourceID;
			arrActiveAlarms[1].iTimeStampCleared := arrEvents[1].iTimeStampCleared;
			arrActiveAlarms[1].iTimeStampConfirmed := arrEvents[1].iTimeStampConfirmed;
			IF iActiveAlarms < iMAX_EVENTS THEN
				iActiveAlarms := iActiveAlarms + 1;
			END_IF
		END_IF
	ELSIF rtAlarmCleard.Q THEN
		//alarmy aktywne
		FOR index := 1 TO iActiveAlarms DO
			IF  GuidsEqualByVal(stBaseEvent.guidEventClass, arrActiveAlarms[index].guidEventClass) AND
				stBaseEvent.iEventId = arrActiveAlarms[index].iEventId AND 
				stBaseEvent.sSourceName = arrActiveAlarms[index].sSourceName AND 
				stBaseEvent.iSourceID = arrActiveAlarms[index].iSourceID THEN
				IF index < iMAX_EVENTS THEN
					MEMCPY(ADR(arrActiveAlarms[index]),ADR(arrActiveAlarms[index+1]),SIZEOF(arrActiveAlarms[1]) * (iActiveAlarms - index));
					MEMSET(ADR(arrActiveAlarms[iActiveAlarms]),0,SIZEOF(arrActiveAlarms[iActiveAlarms]));
					iActiveAlarms := iActiveAlarms - 1;
					EXIT;
				ELSE
					MEMSET(ADR(arrActiveAlarms[iActiveAlarms]),0,SIZEOF(arrActiveAlarms[iActiveAlarms]));
					iActiveAlarms := iActiveAlarms - 1;
				END_IF
			END_IF
		END_FOR
		//alarmy historyczne
		FOR index := 1 TO iMAX_EVENTS DO
			IF  GuidsEqualByVal(stBaseEvent.guidEventClass, arrEvents[index].guidEventClass) AND
				stBaseEvent.iEventId = arrEvents[index].iEventId AND 
				stBaseEvent.sSourceName = arrEvents[index].sSourceName AND 
				stBaseEvent.iSourceID = arrEvents[index].iSourceID THEN
				arrEvents[index].iTimeStampCleared := stBaseEvent.iTimeStamp/10000 - 11644473600000; //100ns to ms -> /1000
				IF NOT bSummertime THEN
					arrEvents[index].iTimeStampCleared := arrEvents[index].iTimeStampCleared + 3600000;
				END_IF
				EXIT;
			END_IF
		END_FOR
	ELSIF stBaseEvent.eEventType = E_EventType.ALARM_CONFIRMED THEN
		FOR index := 1 TO iMAX_EVENTS DO
			IF  GuidsEqualByVal(stBaseEvent.guidEventClass, arrActiveAlarms[index].guidEventClass) AND
				stBaseEvent.iEventId = arrActiveAlarms[index].iEventId AND 
				stBaseEvent.sSourceName = arrActiveAlarms[index].sSourceName AND 
				stBaseEvent.iSourceID = arrActiveAlarms[index].iSourceID THEN
				arrActiveAlarms[index].iTimeStampConfirmed := stBaseEvent.iTimeStamp/10000 - 11644473600000; //100ns to ms -> /1000
				IF NOT bSummertime THEN
					arrActiveAlarms[index].iTimeStampConfirmed := arrActiveAlarms[index].iTimeStampConfirmed + 3600000;
				END_IF
				EXIT;
			END_IF
		END_FOR	
		FOR index := 1 TO iMAX_EVENTS DO
			IF  GuidsEqualByVal(stBaseEvent.guidEventClass, arrEvents[index].guidEventClass) AND
				stBaseEvent.iEventId = arrEvents[index].iEventId AND 
				stBaseEvent.sSourceName = arrEvents[index].sSourceName AND 
				stBaseEvent.iSourceID = arrEvents[index].iSourceID THEN
				arrEvents[index].iTimeStampConfirmed := stBaseEvent.iTimeStamp/10000 - 11644473600000; //100ns to ms -> /1000
				IF NOT bSummertime THEN
					arrEvents[index].iTimeStampConfirmed := arrEvents[index].iTimeStampConfirmed + 3600000;
				END_IF
				EXIT;
			END_IF
		END_FOR	
	END_IF
	
	bReqText := FALSE;
END_IF
END_METHOD

METHOD OnAlarmCleared
VAR_INPUT
	fbEvent : REFERENCE TO FB_TcEvent;
END_VAR
IF iActiveDefinitionEvents >= iMAX_DEFINITION_EVENTS THEN
	RETURN; //skip new events
END_IF

MEMCPY(ADR(arrActiveEvents[2]),ADR(arrActiveEvents[1]),SIZEOF(arrActiveEvents[1]) * iActiveDefinitionEvents);
iActiveDefinitionEvents := iActiveDefinitionEvents + 1;
arrActiveEvents[1].iType := 1;
arrActiveEvents[1].guidEventClass := fbEvent.EventClass;
arrActiveEvents[1].eSeverity := fbEvent.eSeverity;
arrActiveEvents[1].iEventId := fbEvent.nEventId;
arrActiveEvents[1].iTimeStamp := fbEvent.nTimestamp;
arrActiveEvents[1].iTcArguments := fbEvent.ipArguments;
arrActiveEvents[1].eEventType := E_EventType.ALARM_CLEARED;
arrActiveEvents[1].sSourceName := fbEvent.ipSourceInfo.sName;
arrActiveEvents[1].iSourceID := fbEvent.ipSourceInfo.nId;
fbEvent.GetJsonAttribute(arrActiveEvents[1].sJsonAttribute, SIZEOF(arrActiveEvents[1].sJsonAttribute));

(* Active events type counter *)
IF arrActiveEvents[1].eSeverity = TcEventSeverity.Verbose THEN
	IF iActiveInfo > 0 THEN
		iActiveInfo := iActiveInfo - 1;	
	ELSE iActiveInfo :=0;
	END_IF
	
ELSIF arrActiveEvents[1].eSeverity = TcEventSeverity.Info THEN
	IF iActiveVerbose > 0 THEN
		iActiveVerbose := iActiveVerbose - 1;	
	ELSE iActiveVerbose := 0;
	END_IF
ELSIF arrActiveEvents[1].eSeverity = TcEventSeverity.Warning THEN
	IF iActiveWarning > 0 THEN
		iActiveWarning := iActiveWarning - 1;		
	ELSE iActiveWarning := 0;
	END_IF
	
ELSIF arrActiveEvents[1].eSeverity = TcEventSeverity.Error THEN
	IF iActiveError > 0 THEN
		iActiveError := iActiveError - 1;		
	ELSE iActiveError :=0;
	END_IF
	
ELSIF arrActiveEvents[1].eSeverity = TcEventSeverity.Critical THEN
	IF iActiveCritical > 0 THEN
		iActiveCritical := iActiveCritical - 1;	
	ELSE iActiveCritical := 0;
	END_IF
END_IF
END_METHOD

METHOD OnAlarmConfirmed
VAR_INPUT
	fbEvent : REFERENCE TO FB_TcEvent;
END_VAR
IF iActiveDefinitionEvents >= iMAX_DEFINITION_EVENTS THEN
	RETURN; //skip new events
END_IF

MEMCPY(ADR(arrActiveEvents[2]),ADR(arrActiveEvents[1]),SIZEOF(arrActiveEvents[1]) * iActiveDefinitionEvents);
iActiveDefinitionEvents := iActiveDefinitionEvents + 1;
arrActiveEvents[1].iType := 1;
arrActiveEvents[1].guidEventClass := fbEvent.EventClass;
arrActiveEvents[1].eSeverity := fbEvent.eSeverity;
arrActiveEvents[1].iEventId := fbEvent.nEventId;
arrActiveEvents[1].iTimeStamp := fbEvent.nTimestamp;
arrActiveEvents[1].iTcArguments := fbEvent.ipArguments;
arrActiveEvents[1].eEventType := E_EventType.ALARM_CONFIRMED;
arrActiveEvents[1].sSourceName := fbEvent.ipSourceInfo.sName;
arrActiveEvents[1].iSourceID := fbEvent.ipSourceInfo.nId;
fbEvent.GetJsonAttribute(arrActiveEvents[1].sJsonAttribute, SIZEOF(arrActiveEvents[1].sJsonAttribute));

(* Active events type counter *)
IF arrActiveEvents[1].eSeverity = TcEventSeverity.Verbose THEN
	IF iActiveInfo > 0 THEN
		iActiveInfo := iActiveInfo - 1;	
	ELSE 
		iActiveInfo :=0;
	END_IF
		
ELSIF arrActiveEvents[1].eSeverity = TcEventSeverity.Info THEN
	iActiveVerbose := iActiveVerbose - 1;	

ELSIF arrActiveEvents[1].eSeverity = TcEventSeverity.Warning THEN
	IF iActiveWarning > 0 THEN
		iActiveWarning := iActiveWarning - 1;
	ELSE iActiveWarning := 0;
	END_IF
			

ELSIF arrActiveEvents[1].eSeverity = TcEventSeverity.Error THEN
	IF iActiveError > 0 THEN
		iActiveError := iActiveError - 1;
	ELSE iActiveError := 0;	
	END_IF
	
ELSIF arrActiveEvents[1].eSeverity = TcEventSeverity.Critical THEN
	IF iActiveCritical > 0 THEN
		iActiveCritical := iActiveCritical - 1;	
	ELSE iActiveCritical := 0;
	END_IF
END_IF
END_METHOD

METHOD OnAlarmRaised
VAR_INPUT
	fbEvent : REFERENCE TO FB_TcEvent;
END_VAR
VAR
END_VAR
IF iActiveDefinitionEvents >= iMAX_DEFINITION_EVENTS THEN
	RETURN; //skip new events
END_IF

MEMCPY(ADR(arrActiveEvents[2]),ADR(arrActiveEvents[1]),SIZEOF(arrActiveEvents[1]) * iActiveDefinitionEvents);
iActiveDefinitionEvents := iActiveDefinitionEvents + 1;
arrActiveEvents[1].iType := 1;
arrActiveEvents[1].guidEventClass := fbEvent.EventClass;
arrActiveEvents[1].eSeverity := fbEvent.eSeverity;
arrActiveEvents[1].iEventId := fbEvent.nEventId;
arrActiveEvents[1].iTimeStamp := fbEvent.nTimestamp;
arrActiveEvents[1].iTcArguments := fbEvent.ipArguments;
arrActiveEvents[1].eEventType := E_EventType.ALARM_RAISED;
arrActiveEvents[1].sSourceName := fbEvent.ipSourceInfo.sName;
arrActiveEvents[1].iSourceID := fbEvent.ipSourceInfo.nId;
fbEvent.GetJsonAttribute(arrActiveEvents[1].sJsonAttribute, SIZEOF(arrActiveEvents[1].sJsonAttribute));

(* Active events type counter *)
IF arrActiveEvents[1].eSeverity = TcEventSeverity.Verbose THEN
	iActiveInfo := iActiveInfo + 1;	
	
ELSIF arrActiveEvents[1].eSeverity = TcEventSeverity.Info THEN
	IF iActiveVerbose < 4294967295 THEN
		iActiveVerbose := iActiveVerbose + 1;	
	ELSE iActiveVerbose := 4294967295;
	END_IF
	
ELSIF arrActiveEvents[1].eSeverity = TcEventSeverity.Warning THEN
	IF iActiveWarning < 4294967295 THEN
		iActiveWarning := iActiveWarning + 1;	
	ELSE iActiveWarning := 4294967295;
	END_IF
	
ELSIF arrActiveEvents[1].eSeverity = TcEventSeverity.Error THEN
	IF iActiveError < 4294967295 THEN
		iActiveError := iActiveError + 1;	
	ELSE iActiveError := 4294967295;
	END_IF
	
ELSIF arrActiveEvents[1].eSeverity = TcEventSeverity.Critical THEN
	IF iActiveCritical < 4294967295 THEN
		iActiveCritical := iActiveCritical + 1;	
	ELSE iActiveCritical := 4294967295;
	END_IF
	
END_IF
END_METHOD

METHOD OnMessageSent
VAR_INPUT
	fbEvent : REFERENCE TO FB_TcEvent;
END_VAR

VAR 
END_VAR
IF iActiveDefinitionEvents >= iMAX_DEFINITION_EVENTS THEN
	RETURN; //skip new events
END_IF

MEMCPY(ADR(arrActiveEvents[2]),ADR(arrActiveEvents[1]),SIZEOF(arrActiveEvents[1]) * iActiveDefinitionEvents);
iActiveDefinitionEvents := iActiveDefinitionEvents + 1;
arrActiveEvents[1].iType := 2;
arrActiveEvents[1].guidEventClass := fbEvent.EventClass;
arrActiveEvents[1].eSeverity := fbEvent.eSeverity;
arrActiveEvents[1].iEventId := fbEvent.nEventId;
arrActiveEvents[1].iTimeStamp := fbEvent.nTimestamp;
arrActiveEvents[1].iTcArguments := fbEvent.ipArguments;
arrActiveEvents[1].eEventType := E_EventType.MESSAGE;
arrActiveEvents[1].sSourceName := fbEvent.ipSourceInfo.sName;
arrActiveEvents[1].iSourceID := fbEvent.ipSourceInfo.nId;
fbEvent.GetJsonAttribute(arrActiveEvents[1].sJsonAttribute, SIZEOF(arrActiveEvents[1].sJsonAttribute));
END_METHOD

END_FUNCTION_BLOCK

// ---- POUs/Machine/FB_MachineSafety.TcPOU
FUNCTION_BLOCK FB_MachineSafety EXTENDS FB_UniversalSafety
VAR
	bRunStop 						AT %Q* 	: BOOL;
	bErrorACK 						AT %Q* 	: BOOL;
	bFB_Error 						AT %I* 	: BOOL;
	bComm_Error 					AT %I* 	: BOOL;
	                                       	
	bRestartButton 					AT %I* 	: BOOL;
	bPressureEDM 					AT %I* 	: BOOL;
	bEStopContactorsEDM 			AT %I* 	: BOOL;
	bCoverContactorsEDM 			AT %I* 	: BOOL;
	bTrayHandlerContactorsEDM 		AT %I* 	: BOOL;
	                                       	
	bRestartButtonOut 				AT %Q* 	: BOOL;
	bPressureEDMOut 				AT %Q* 	: BOOL;
	bEStopContactorsEDMOut			AT %Q* 	: BOOL;
	bCoverContactorsEDMOut 			AT %Q* 	: BOOL;
	bTrayHandlerContactorsEDMOut 	AT %Q*	: BOOL;
	
	piInputSafeDataE_StopA					: FB_DigitalInput;
	piInputSafeDataE_StopB					: FB_DigitalInput;
	piInputSafeDataSafetyOverrideA			: FB_DigitalInput;
	piInputSafeDataSafetyOverrideB			: FB_DigitalInput;
	
	piInputSafeDataDoorLockA				: FB_DigitalInput;
	piInputSafeDataDoorLockB				: FB_DigitalInput;
	piInputSafeDataRobotE_StopA				: FB_DigitalInput;
	piInputSafeDataRobotE_StopB				: FB_DigitalInput;
	
	piInputSafeDataExternalE_StopA			: FB_DigitalInput;
	piInputSafeDataExternalE_StopB			: FB_DigitalInput;
	piInputSafeDataTrayFeederCourtainA		: FB_DigitalInput;
	piInputSafeDataTrayFeederCourtainB		: FB_DigitalInput;
	
	piInputSafeDataSlowStartValve			: FB_DigitalInput;
	piInputSafeDataE_StopContactor			: FB_DigitalInput;
	piInputSafeDataCoverContactors			: FB_DigitalInput;
	piInputSafeDataTrayHandlerContactors	: FB_DigitalInput;
	
	bE_Stop									: BOOL;
	bSafetyOverride 						: BOOL;
	bDoorLock								: BOOL;
	bRobotE_Stop							: BOOL;
	bExternalE_Stop 						: BOOL;
	bTrayfeederCourtain						: BOOL;
	bSlowStartValve							: BOOL;
	bE_StopContactor						: BOOL;
	bCoverContactors						: BOOL;
	bTrayfeederContactors					: BOOL;
	
END_VAR

(* Send EDM data from standard inputs to Safety Program *)
bCoverContactorsEDMOut 			:= bCoverContactorsEDM;
bEStopContactorsEDMOut 			:= bEStopContactorsEDM;
bPressureEDMOut 				:= bPressureEDM;
bTrayHandlerContactorsEDMOut 	:= bTrayHandlerContactorsEDM;
bRestartButtonOut 				:= bRestartButton;

(* Run parent *)
SUPER^();

(* Refresh data from Safe Logic Module *)
piInputSafeDataE_StopA();
piInputSafeDataE_StopB();
piInputSafeDataSafetyOverrideA();
piInputSafeDataSafetyOverrideB();

piInputSafeDataDoorLockA();
piInputSafeDataDoorLockB();
piInputSafeDataRobotE_StopA();
piInputSafeDataRobotE_StopB();

piInputSafeDataExternalE_StopA();
piInputSafeDataExternalE_StopB();
piInputSafeDataTrayFeederCourtainA();
piInputSafeDataTrayFeederCourtainB();

piInputSafeDataSlowStartValve();
piInputSafeDataE_StopContactor();
piInputSafeDataCoverContactors();
piInputSafeDataTrayHandlerContactors();

(* Update status for PLC program *)
bE_Stop 				:= piInputSafeDataE_StopA.In AND piInputSafeDataE_StopB.In;
bSafetyOverride 		:= piInputSafeDataSafetyOverrideA.In AND piInputSafeDataSafetyOverrideB.In;
bDoorLock 				:= piInputSafeDataDoorLockA.In AND piInputSafeDataDoorLockB.In;
bRobotE_Stop 			:= piInputSafeDataRobotE_StopA.In AND piInputSafeDataRobotE_StopB.In;
bExternalE_Stop 		:= piInputSafeDataExternalE_StopA.In AND piInputSafeDataExternalE_StopB.In;
bTrayfeederCourtain 	:= piInputSafeDataTrayFeederCourtainA.In AND piInputSafeDataTrayFeederCourtainB.In;

(* Used to trigger state change -> Emergency *)
bSlowStartValve 		:= piInputSafeDataSlowStartValve.In;
bE_StopContactor		:= piInputSafeDataE_StopContactor.In;
bCoverContactors		:= piInputSafeDataCoverContactors.In;
bTrayfeederContactors	:= piInputSafeDataTrayHandlerContactors.In;

PROPERTY Comm_Error : BOOL
GET
Comm_Error := bComm_Error;
END_GET
END_PROPERTY

PROPERTY CoverContactors : REFERENCE TO BOOL
GET
CoverContactors REF= bCoverContactors;
END_GET
END_PROPERTY

PROPERTY CoverContactorsEDM : BOOL
GET
CoverContactorsEDM := bCoverContactorsEDM;
END_GET
END_PROPERTY

PROPERTY DoorLock : REFERENCE TO BOOL
GET
DoorLock REF= bDoorLock;
END_GET
END_PROPERTY

PROPERTY E_Stop : REFERENCE TO BOOL
GET
E_Stop REF= bE_Stop;
END_GET
END_PROPERTY

PROPERTY E_StopContactors : REFERENCE TO BOOL
GET
E_StopContactors REF= bE_StopContactor;
END_GET
END_PROPERTY

PROPERTY ErrorAck : BOOL
GET
ErrorAck := bErrorACK;
END_GET
SET
bErrorACK := ErrorAck;
END_SET
END_PROPERTY

PROPERTY EStopContactorsEDM : BOOL
GET
EStopContactorsEDM := bEStopContactorsEDM;
END_GET
END_PROPERTY

PROPERTY ExternalE_Stop : REFERENCE TO BOOL
GET
ExternalE_Stop REF= bExternalE_Stop;
END_GET
END_PROPERTY

PROPERTY FB_Error : BOOL
GET
FB_Error := bFB_Error;
END_GET
END_PROPERTY

METHOD MR_Abort : BOOL
VAR_INPUT
END_VAR
END_METHOD

METHOD MR_FirstCycle : BOOL
VAR_INPUT
END_VAR
END_METHOD

METHOD MR_Init : BOOL
VAR_INPUT
END_VAR
END_METHOD

METHOD MR_Reset : BOOL
VAR_INPUT
END_VAR
END_METHOD

METHOD PROTECTED MS_Aborting
VAR_INPUT
END_VAR
;
END_METHOD

METHOD PROTECTED MS_Initializing
VAR_INPUT
END_VAR
;
END_METHOD

METHOD PROTECTED MS_ReadyInitialized
VAR_INPUT
END_VAR
;
END_METHOD

METHOD PROTECTED MS_Reset
VAR_INPUT
END_VAR
END_METHOD

METHOD PROTECTED MS_ResetDone
VAR_INPUT
END_VAR
END_METHOD

METHOD PROTECTED MS_Running
VAR_INPUT
END_VAR
;
END_METHOD

METHOD PROTECTED MS_Uninitialized
VAR_INPUT
END_VAR
;
END_METHOD

PROPERTY PressureEDM : BOOL
GET
PressureEDM := bPressureEDM;
END_GET
END_PROPERTY

PROPERTY ref_InputSafeDataCoverContactors : REFERENCE TO FB_DigitalInput
GET
ref_InputSafeDataCoverContactors REF= piInputSafeDataCoverContactors;
END_GET
END_PROPERTY

PROPERTY ref_InputSafeDataDoorLockA : REFERENCE TO FB_DigitalInput
GET
ref_InputSafeDataDoorLockA REF= piInputSafeDataDoorLockA;
END_GET
END_PROPERTY

PROPERTY ref_InputSafeDataDoorLockB : REFERENCE TO FB_DigitalInput
GET
ref_InputSafeDataDoorLockB REF= piInputSafeDataDoorLockB;
END_GET
END_PROPERTY

PROPERTY ref_InputSafeDataE_StopA : REFERENCE TO FB_DigitalInput
GET
ref_InputSafeDataE_StopA REF= piInputSafeDataE_StopA;
END_GET
END_PROPERTY

PROPERTY ref_InputSafeDataE_StopB : REFERENCE TO FB_DigitalInput
GET
ref_InputSafeDataE_StopB REF= piInputSafeDataE_StopB;
END_GET
END_PROPERTY

PROPERTY ref_InputSafeDataE_StopContactor : REFERENCE TO FB_DigitalInput
GET
ref_InputSafeDataE_StopContactor REF= piInputSafeDataE_StopContactor;
END_GET
END_PROPERTY

PROPERTY ref_InputSafeDataExternalE_StopA : REFERENCE TO FB_DigitalInput
GET
ref_InputSafeDataExternalE_StopA REF= piInputSafeDataExternalE_StopA;
END_GET
END_PROPERTY

PROPERTY ref_InputSafeDataExternalE_StopB : REFERENCE TO FB_DigitalInput
GET
ref_InputSafeDataExternalE_StopB REF= piInputSafeDataExternalE_StopB;
END_GET
END_PROPERTY

PROPERTY ref_InputSafeDataRobotE_StopA : REFERENCE TO FB_DigitalInput
GET
ref_InputSafeDataRobotE_StopA REF= piInputSafeDataRobotE_StopA;
END_GET
END_PROPERTY

PROPERTY ref_InputSafeDataRobotE_StopB : REFERENCE TO FB_DigitalInput
GET
ref_InputSafeDataRobotE_StopB REF= piInputSafeDataRobotE_StopB;
END_GET
END_PROPERTY

PROPERTY ref_InputSafeDataSafetyOverrideA : REFERENCE TO FB_DigitalInput
GET
ref_InputSafeDataSafetyOverrideA REF= piInputSafeDataSafetyOverrideA;
END_GET
END_PROPERTY

PROPERTY ref_InputSafeDataSafetyOverrideB : REFERENCE TO FB_DigitalInput
GET
ref_InputSafeDataSafetyOverrideB REF= piInputSafeDataSafetyOverrideB;
END_GET
END_PROPERTY

PROPERTY ref_InputSafeDataSlowStartValve : REFERENCE TO FB_DigitalInput
GET
ref_InputSafeDataSlowStartValve REF= piInputSafeDataSlowStartValve;
END_GET
END_PROPERTY

PROPERTY ref_InputSafeDataTrayfeederContactors : REFERENCE TO FB_DigitalInput
GET
ref_InputSafeDataTrayfeederContactors REF= piInputSafeDataTrayHandlerContactors;
END_GET
END_PROPERTY

PROPERTY ref_InputSafeDataTrayfeederCourtainA : REFERENCE TO FB_DigitalInput
GET
ref_InputSafeDataTrayfeederCourtainA REF= piInputSafeDataTrayFeederCourtainA;
END_GET
END_PROPERTY

PROPERTY ref_InputSafeDataTrayfeederCourtainB : REFERENCE TO FB_DigitalInput
GET
ref_InputSafeDataTrayfeederCourtainB REF= piInputSafeDataTrayFeederCourtainB;
END_GET
END_PROPERTY

PROPERTY RestartButton : BOOL
GET
RestartButton := bRestartButton;
END_GET
END_PROPERTY

PROPERTY RobotE_Stop : REFERENCE TO BOOL
GET
RobotE_Stop REF= bRobotE_Stop;
END_GET
END_PROPERTY

PROPERTY RunStop : BOOL
GET
RunStop := bRunStop;
END_GET
SET
bRunStop := RunStop;
END_SET
END_PROPERTY

PROPERTY SafetyOverride : REFERENCE TO BOOL
GET
SafetyOverride REF= bSafetyOverride;
END_GET
END_PROPERTY

PROPERTY SlowStartValveContactors : REFERENCE TO BOOL
GET
SlowStartValveContactors REF= bSlowStartValve;
END_GET
END_PROPERTY

PROPERTY TrayfeederContactors : REFERENCE TO BOOL
GET
TrayfeederContactors REF= bTrayfeederContactors;
END_GET
END_PROPERTY

PROPERTY TrayfeederContactorsEDM : BOOL
GET
TrayfeederContactorsEDM := bTrayHandlerContactorsEDM;
END_GET
END_PROPERTY

PROPERTY TrayfeederCourtain : REFERENCE TO BOOL
GET
TrayfeederCourtain REF= bTrayfeederCourtain;
END_GET
END_PROPERTY

END_FUNCTION_BLOCK

// ---- POUs/PRG/PRG_FB_BowlFeeder.TcPOU
PROGRAM PRG_FB_BowlFeeder
VAR
	bFirstCycle 			: BOOL := TRUE;
	fbBowlFeeder 			: FB_BowlFeeder;
	
	rSetSp	: REAL := 50;

	bInit 					: BOOL;
	bAbort 					: BOOL;
	bReset					: BOOL;
	bStart					: BOOL;
	bStop					: BOOL;

	bActive					: BOOL;
	bRunning				: BOOL;
	bError					: BOOL;
	iErrorID				: UDINT;
	

	rSetpoint: REAL;
END_VAR

(* Setting initial parameters *)
IF bFirstCycle THEN
	bFirstCycle := FALSE;
	
	fbBowlFeeder.MR_FirstCycle(sName := 'Bowl Feeder');
	fbBowlFeeder.Setpoint := rSetSp;
END_IF

bActive := fbBowlFeeder.Active;
bRunning := fbBowlFeeder.Running;
bError := fbBowlFeeder.Error;
rSetpoint := fbBowlFeeder.Setpoint;

(* Simple controler *)
IF bInit THEN
	fbBowlFeeder.MR_Init();
	IF fbBowlFeeder.Active THEN
		bInit := FALSE;
	END_IF
END_IF

IF bStart THEN
	fbBowlFeeder.MR_Start();
	IF fbBowlFeeder.Running THEN
 		bStart := FALSE;
	END_IF
END_IF

IF bStop THEN
	fbBowlFeeder.MR_Stop();
	IF NOT fbBowlFeeder.Running THEN
 		bStop := FALSE;
	END_IF
END_IF

fbBowlFeeder();

END_PROGRAM

// ---- POUs/PRG/PRG_MachineSafety.TcPOU
PROGRAM PRG_MachineSafety
VAR
	bFirstCycle 	: BOOL := TRUE;
	fbMachineSafety : FB_MachineSafety;
END_VAR

(* First cycle of visu controler run*)
IF bFirstCycle THEN
	bFirstCycle := FALSE;
	
	(* Assign machine controler reference to Shell API*)
	stShell.stPlatform.ref_MachineSafety REF= fbMachineSafety;
	
END_IF

(* Cyclic run of machine safety *)
fbMachineSafety();

END_PROGRAM

// ---- GlobalTextList.TcGTLO
TEXTLIST GlobalTextList
  150 = '%2.1f'
  250 = '%2.2f'
  1258 = '%2.4f'
  224 = '%2d'
  1044 = '%3.0f'
  1573 = '%3.1f'
  21 = '%6.3f'
  331 = '%d'
  890 = '%f'
  1627 = '%ms'
  976 = '%s'
  361 = "%t[s's']"
  2692 = '%t[s]'
  2051 = '/'
  887 = 'Abort'
  494 = 'Acceleration:'
  3798 = 'Action number:'
  487 = 'Active Alarms'
  1711 = 'Active alarms:'
  649 = 'Active critical'
  1670 = 'Active critical alarms:'
  202 = 'Active criticals:'
  709 = 'Active errors'
  780 = 'Active errors:'
  700 = 'Active warnings:'
  582 = 'Active warrnings'
  706 = 'Active warrnings:'
  370 = 'Actual Position:'
  78 = 'Actual Velocity'
  1000 = 'Admin'
  431 = 'Alarms'
  813 = 'All active alarms:'
  944 = 'At least one of emergency button is active'
  1158 = 'At least one of the door lock is not locked'
  427 = 'Auto mode'
  989 = 'Auxilary'
  931 = 'Axes'
  913 = 'Axis'
  542 = 'Back'
  300 = 'Backup'
  2292 = 'Backup and restore from external directory'
  2866 = 'Batch Data'
  2617 = 'Batch ID'
  2549 = 'Batch Performance'
  1008 = 'Batch Settings'
  2272 = 'Battery low'
  662 = 'Battery reset'
  161 = 'Bowl Feeder'
  1355 = 'Camera'
  576 = 'Camera connection'
  2594 = 'Camera Focus\nCheck'
  564 = 'Camera Focus Check'
  2601 = 'Camera job setup'
  917 = 'Change pass.'
  1549 = 'Clear all'
  349 = 'Clear All Alarms'
  277 = 'Close'
  410 = 'Close HMI'
  1072 = 'Commands'
  186 = 'Communication Setup'
  1536 = 'Complete'
  592 = 'Continue'
  1156 = 'Controller'
  2906 = 'Controller reset'
  470 = "Couldn't connect to any measurement setup"
  3304 = "Couldn't connect to measurement setup"
  1448 = 'Courtains checked'
  1047 = 'Create'
  2909 = 'Create new recipe:'
  3176 = 'Current state:'
  2120 = 'Current value'
  2043 = 'Cycle pause'
  3558 = 'Cycle restore'
  2070 = 'Cycle stop'
  424 = 'Cylinders'
  1092 = 'Deceleration:'
  362 = 'Deinitialization in progress...'
  115 = 'Delay '
  301 = 'Dent'
  1655 = 'Digital Inputs'
  1456 = 'Digital inputs'
  1692 = 'Digital Outputs'
  1445 = 'Digital outputs'
  1090 = 'Digital outputs and valves'
  2518 = 'Dirt'
  1004 = 'Distance'
  538 = 'Door Lock'
  1033 = 'Door locks checked'
  2366 = 'E-Stop checked'
  956 = 'Enable'
  1643 = 'Enable simulation'
  245 = 'Enable/Disable All'
  1468 = 'Error'
  2495 = 'Error inform'
  2782 = 'Error reset'
  537 = 'Error: %d'
  1738 = 'Error: %s'
  368 = 'Event history'
  1107 = 'Event history:'
  86 = 'Event ID'
  619 = 'Event Text'
  297 = 'Event Type'
  77 = 'Export to file'
  1865 = 'File name'
  2449 = 'File Name:'
  1073 = 'Finishing initialization...'
  742 = 'Fixture 1'
  433 = 'Fixture 2'
  643 = 'Fixture 3'
  801 = 'Fixture 4'
  404 = 'Fixture 5'
  945 = 'Fixture 6'
  230 = 'Fixture 7'
  591 = 'Fixture 8'
  1032 = 'Fixture initialization (1)'
  526 = 'Fixture initialization (2)'
  708 = 'Fixture initialization (3)'
  710 = 'Fixture initialization (4)'
  416 = 'Fixture initialization (5)'
  888 = 'Fixture initialization (6)'
  738 = 'Fixture initialization (7)'
  405 = 'Fixture initialization (8)'
  1696 = 'Force Input Value'
  2573 = 'General FCQ State:'
  244 = 'Go %s'
  2687 = 'Go auto'
  66 = 'Go home'
  29 = 'Golden Sample'
  2114 = 'Golden Sample\nCheck'
  2384 = 'Good'
  440 = 'Good Blow Time'
  2052 = 'Good Distance'
  274 = 'Good Position'
  70 = 'Good quantity'
  182 = 'GS Type'
  1163 = 'Halt'
  2141 = 'Halted'
  110 = 'Home'
  1505 = 'Homed'
  2548 = 'In Position'
  371 = 'Initialize'
  1488 = 'Initialized'
  2081 = 'Input Quality'
  312 = 'Inputs'
  1273 = 'IP Address'
  2436 = 'Jog'
  18 = 'Jog +'
  19 = 'Jog -'
  2152 = 'Jog mode:'
  121 = 'Lag error:'
  715 = 'Lights'
  1263 = 'Load from file'
  546 = 'Load from Recipes'
  1426 = 'Loaded recipe'
  3542 = 'Local path'
  2198 = 'Lock'
  1750 = 'Lock the doors before going back to full speed'
  332 = 'Log In'
  198 = 'Log Out'
  1506 = 'Logged user'
  466 = 'Machine Initial Setup'
  1379 = 'Machine Initial Startup'
  507 = 'Machine Logger initialization'
  921 = 'Machine nearly ready to work...'
  665 = 'Machine state'
  428 = 'Manual'
  485 = 'Manual Axis Control'
  1020 = 'Manual Cylinders Control'
  822 = 'Manual mode'
  3024 = 'Manual Robots Control'
  83 = 'Measurement fixtures setup'
  67 = 'MES connection'
  2665 = 'MES delay'
  644 = 'MES file command dwell time:'
  729 = 'Mode switch'
  417 = 'Motors'
  1606 = 'Next'
  1295 = 'No dry run'
  1023 = 'None'
  616 = 'Normfile-Config'
  1645 = 'Number of:'
  1015 = 'Operator'
  1972 = 'Others'
  1697 = 'Output trays replaced'
  613 = 'Outputs'
  639 = 'Override:'
  1319 = 'Override: %2.0d'
  407 = 'Override: %2d'
  1429 = 'Override: %3.0f'
  1146 = 'Parameters:'
  1309 = 'Path:'
  2305 = 'Pause'
  725 = 'Paused'
  3825 = 'Pick&Place Only'
  2613 = 'Place empty trays inside machine output zone and close the cover'
  1304 = 'Port'
  93 = 'Position'
  1845 = 'Position hold'
  2517 = 'Position:'
  905 = 'Position: %s'
  731 = 'Powered on'
  1584 = 'Press " Safety Reset" button at front panel'
  1825 = 'Previous'
  3063 = 'Product Item-Config'
  2388 = 'Production Order (PO)'
  316 = 'Program'
  1005 = 'Read to file'
  1949 = 'Recipe'
  690 = 'Recipe list:'
  2365 = 'Recipe name'
  1499 = 'Recipe name:'
  247 = 'Recipe parameters'
  298 = 'Recipes'
  260 = 'Recipes Manager initialization'
  2656 = 'Recipes Manager: %s'
  2461 = 'Reduced Speed'
  1796 = 'Reject'
  647 = 'Rejected quantity'
  1083 = 'Release'
  2097 = 'Reload'
  3410 = 'Remote path'
  2954 = 'Remove'
  3075 = 'Reset'
  707 = 'Reset in progress...'
  861 = 'Reset:'
  1061 = 'Reseting errors...'
  561 = 'Restore'
  2648 = 'Restore auto'
  854 = 'Retry'
  2957 = 'Rework'
  1951 = 'Rework Processing'
  1759 = 'Rework quantity'
  610 = 'Robot 1'
  704 = 'Robot Controlers Communication Setup'
  1558 = 'Robot Controlers Power On ( aprox. 60 sec.)'
  1027 = 'Robot Controlers reset'
  1702 = 'Robot homed'
  2693 = 'Robot homed (1)'
  2286 = 'Robot homed (2)'
  590 = 'Robot initialization'
  155 = 'Robot initialization (1)'
  1178 = 'Robot initialization (2)'
  951 = 'Robots'
  463 = 'Robots Controler Power On'
  2245 = 'Robots in automatic mode'
  1226 = 'Robots in remote mode'
  1611 = 'Rotary table'
  1886 = 'Rotary table homed'
  962 = 'Rotary table initialization'
  2099 = 'RTC Vision'
  3103 = 'RTC Vision System'
  2584 = 'Safe Inputs'
  958 = 'Safe mode switch in progress...'
  711 = 'Safe mode switching...'
  1087 = 'Safe Outputs'
  2044 = 'Safety Controler check'
  2118 = 'Safety Controler initialization'
  1398 = 'Safety Controler reset'
  980 = 'Safety Controler start'
  670 = 'Safety I/O'
  1981 = 'Sample ID'
  556 = 'Samples measured: %d'
  2626 = 'Save in file'
  550 = 'Select'
  1288 = 'Selected recipe'
  7 = 'Selected recipe value'
  1458 = 'Selected recipe:'
  1007 = 'Service'
  2402 = 'Servo off'
  772 = 'Servo on'
  2183 = 'Set Position:'
  511 = 'Set Velocity:'
  916 = 'Setpoint'
  536 = 'Severity'
  2362 = 'Skip to next'
  1781 = 'Skip tray change'
  50 = 'Software version: v%s'
  1856 = 'Sort Good Blow Time'
  959 = 'Sort Good Distance'
  1950 = 'Sort Station Parameters'
  820 = 'Sorting Station'
  562 = 'Sorting Station Parameter'
  827 = 'SP'
  450 = 'Start'
  2048 = 'START'
  3789 = 'Started'
  1037 = 'State: %s'
  895 = 'Status'
  85 = 'Statuses & parameters:'
  442 = 'Stop'
  563 = 'STOP'
  1093 = 'Stopped'
  2590 = 'Time'
  359 = 'Time (s)'
  848 = 'Time Cleared'
  730 = 'Time Confirmed'
  9 = 'Time Raised'
  1974 = 'Time: %d [ms]'
  10 = 'Total active alarms'
  411 = 'Tray ID'
  3571 = 'Trayfeeder courtain signal interupted'
  3 = 'Trayfeeder courtain signal interupted while initialization'
  109 = 'Trayfeeder home'
  513 = 'Trayfeeder initialization'
  1629 = 'Update recipes'
  1902 = 'Use Adapter'
  1832 = 'UTU 1'
  458 = 'UTU 2'
  124 = 'UTU 3'
  800 = 'UTU 4'
  236 = 'UTU 5'
  779 = 'UTU 6'
  59 = 'UTU 7'
  687 = 'UTU 8'
  342 = 'UTU Device 1'
  668 = 'UTU Device 2'
  5 = 'UTU Device 3'
  1708 = 'UTU Device 4'
  1132 = 'UTU Device 5'
  48 = 'UTU Device 6'
  1515 = 'UTU Device 7'
  948 = 'UTU Device 8'
  1334 = 'Velocity:'
  2437 = 'Vision system'
  322 = '[%s/s]'
  374 = '[%s]'
END_TEXTLIST

// ---- VISUs/Headers/Header.TcVIS
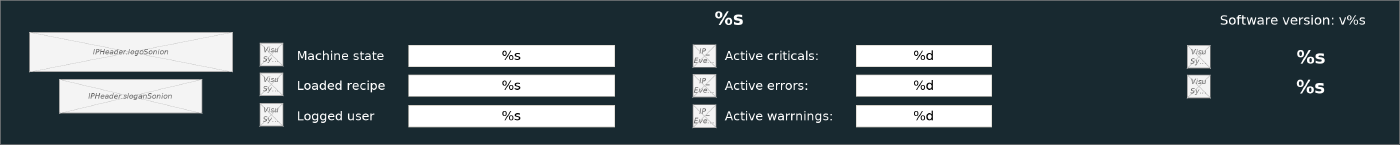
VISUALIZATION Header  // 1920x200
VAR_IN_OUT
	sMachineName		: STRING;					(*  *)
	sSoftwareVersion	: STRING;					(*  *)
	eMachineState		: E_MachineCtrlState;		(*  *)
	sCurrentRecipe		: STRING;					(*  *)
	sCurrentUser		: STRING;					(*  *)
	iActiveCriticals 	: UDINT;					(*  *)
	iActvieErrors		: UDINT;					(*  *)
	iActiveWarrnings	: UDINT;					(*  *)
	sCurrentDate		: STRING;					(*  *)
	sCurrentTime		: STRING;					(*  *)
END_VAR
    Label (404,59 133x36), "Machine state"
    Textfield (560,62 283x30), "%s", text list: 'TL_HeaderMachineState', text index: eMachineState
    Label (404,100 133x36), "Loaded recipe"
    Textfield (560,103 283x30), "%s", text variable: sCurrentRecipe
    Label (404,142 133x36), "Logged user"
    Textfield (560,145 283x30), "%s", text variable: sCurrentUser, text list: ''
    Label (991,59 133x36), "Active criticals:"
    Label (991,100 133x36), "Active errors:"
    Label (991,142 171x36), "Active warrnings:"
    Textfield (1174,62 186x30), "%d", text variable: iActiveCriticals
    Textfield (1174,103 186x30), "%d", text variable: iActvieErrors
    Textfield (1174,145 186x30), "%d", text variable: iActiveWarrnings
    Image (950,61 32x32), image: IP_EventSeverity.critical
    Image (950,102 32x32), image: IP_EventSeverity.error
    Image (950,144 32x32), image: IP_EventSeverity.warning
    Image (1628,62 32x32), image: VisuSymbols.Symbols.Calender
    Image (1628,103 32x32), image: VisuSymbols.Symbols.Clock
    Image (356,142 32x32), image: VisuSymbols.Symbols.User
    Image (356,59 32x32), image: VisuSymbols.Symbols.voltage
    Image (356,100 32x32), image: VisuSymbols.Symbols.Doc
    Textfield (700,10 600x30), "%s", text variable: sMachineName
    Textfield (1670,10 250x36), "Software version: v%s", text variable: sSoftwareVersion
    Textfield (1692,62 212x33), "%s", text variable: sCurrentDate
    Textfield (1691,103 213x33), "%s", text variable: sCurrentTime
    Image (40,44 279x55), image: IPHeader.logoSonion
    Image (81,109 196x47), image: IPHeader.sloganSonion
END_VISUALIZATION

// ---- VISUs/Main.TcVIS
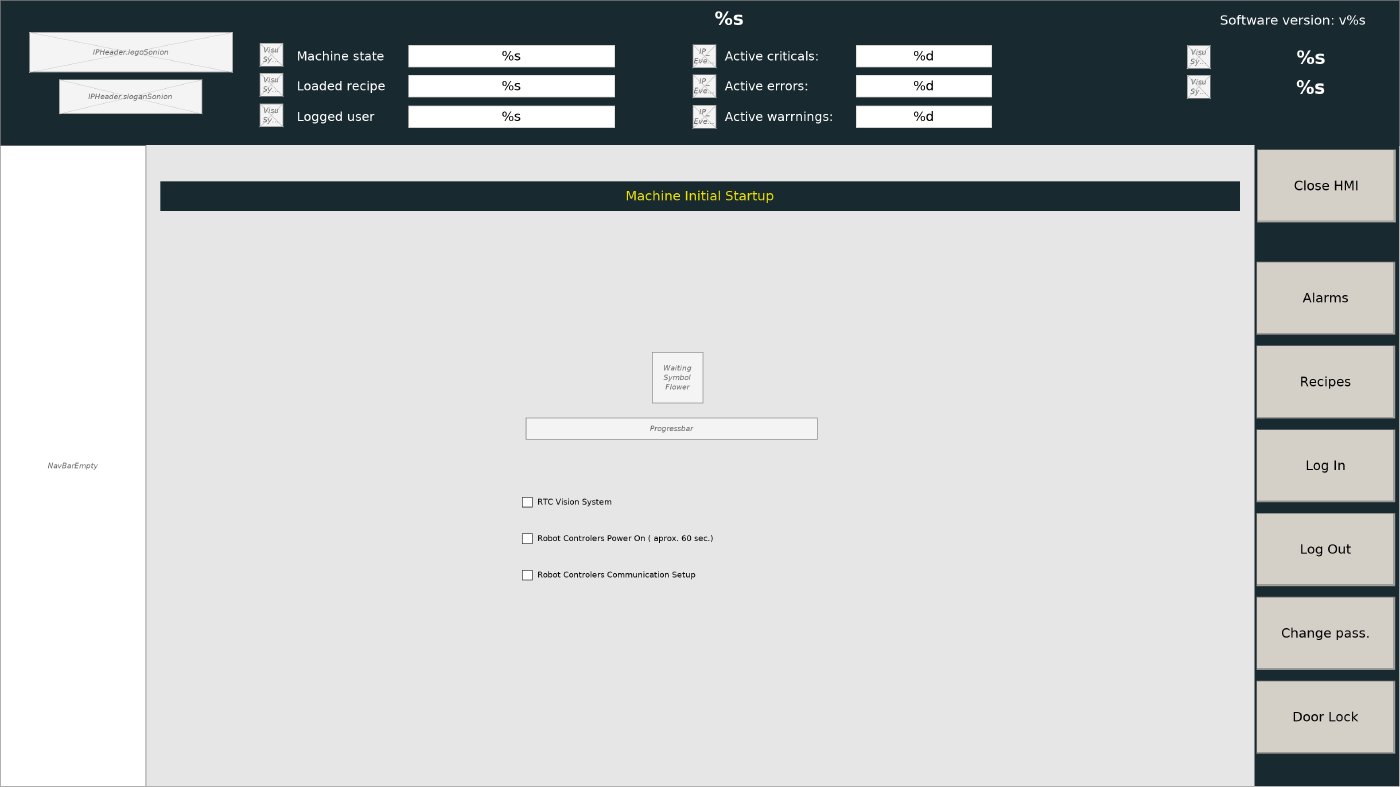
VISUALIZATION Main  // 1920x1080
    Frame (0,0 1920x200)
        shows Header(sMachineName := PRG_VisuControl.fbVisuControl.sMachineName, sSoftwareVersion := PRG_VisuControl.fbVisuControl.sSoftwareVersion, eMachineState := PRG_MachineControl.fbMachineControler.eMachineState, sCurrentRecipe := PRG_VisuControl.fbVisuControl.sCurrentRecipe, sCurrentUser := PRG_VisuControl.fbVisuControl.sCurrentUser, iActiveCriticals := PRG_VisuControl.fbVisuControl.iActiveCriticals, iActvieErrors := PRG_VisuControl.fbVisuControl.iActvieErrors, iActiveWarrnings := PRG_VisuControl.fbVisuControl.iActiveWarrnings, sCurrentDate := PRG_VisuControl.fbVisuControl.sCurrentDate, sCurrentTime := PRG_VisuControl.fbVisuControl.sCurrentTime)
    Frame (1719,199 200x880)
        shows NavBarAuxilary(btnAlarms := PRG_VisuControl.fbVisuControl.btnAlarms, btnRecipes := PRG_VisuControl.fbVisuControl.btnRecipes, btnDoorLock := PRG_VisuControl.fbVisuControl.btnLights, btnLogIn := PRG_VisuControl.fbVisuControl.btnLogIn, btnLogOut := PRG_VisuControl.fbVisuControl.btnLogOut, btnHmiClose := PRG_VisuControl.fbVisuControl.btnHmiClose, sCloseHMIFileName := PRG_VisuControl.fbVisuControl.sCloseHMIFileName, sCloseHMIParameters := PRG_VisuControl.fbVisuControl.sCloseHMIParameters, bVisNotInit := PRG_VisuControl.fbVisuControl.bVisNotInit, bVisHmiCLose := PRG_VisuControl.fbVisuControl.bVisHmiClose, bVisLogIn := PRG_VisuControl.fbVisuControl.bVisLogIn, bVisLogOut := PRG_VisuControl.fbVisuControl.bVisLogOut, bDoorLockDisabled := PRG_VisuControl.fbVisuControl.btnLights, bDoorLockInvisible := PRG_VisuControl.fbVisuControl.btnLights)
    Frame (200,199 1520x880), frame switch variable: PRG_VisuControl.fbVisuControl.eCurrentScreen
        shows PageUninitialized()
        shows PageInitializing(iProgressBar := PRG_VisuControl.fbVisuControl.iInitProgressBar)
        shows PageReadyInitialized()
        shows PageAuto()
        shows PageSwitchMode()
        shows PageManualRobots(btnPrevious := PRG_VisuControl.fbVisuControl.btnPrevious, btnNext := PRG_VisuControl.fbVisuControl.btnNext, bPreviousInvisible := PRG_VisuControl.fbVisuControl.bPreviousInvisible, bNextInvisible := PRG_VisuControl.fbVisuControl.bNextInvisible, stRobotEmpty := PRG_VisuControl.fbVisuControl.arrRobotFrameEmpty[PRG_VisuControl.fbVisuControl.iSelectedRobotPageIndex], stRobot := PRG_VisuControl.fbVisuControl.arrRobotFrame[PRG_VisuControl.fbVisuControl.iSelectedRobotPageIndex], iRobotSelectedPageIndex := PRG_VisuControl.fbVisuControl.iSelectedRobotPageIndex, iRobotTotalPageIndex := PRG_VisuControl.fbVisuControl.iRobotPageIndex)
        shows PageAborting()
        shows PageAlarms(btnClearAllAlarms := PRG_VisuControl.fbVisuControl.btnClearAll, btnExportEvents := PRG_VisuControl.fbVisuControl.btnExport, iActiveAlarms := PRG_VisuControl.fbVisuControl.iActiveAlarms, iActiveCritical := PRG_VisuControl.fbVisuControl.iActiveCriticals, iActiveErrors := PRG_AlarmControl.fbAlarmControler.iActiveError, iActiveWarrnings := PRG_VisuControl.fbVisuControl.iActiveWarrnings, arrEvents := PRG_AlarmControl.fbAlarmControler.EventsTable, arrAlarms := PRG_AlarmControl.fbAlarmControler.AlarmsTable)
        shows PageManualAxis(btnPrevious := PRG_VisuControl.fbVisuControl.btnPrevious, btnNext := PRG_VisuControl.fbVisuControl.btnNext, bPreviousInvisible := PRG_VisuControl.fbVisuControl.bPreviousInvisible, bNextInvisible := PRG_VisuControl.fbVisuControl.bNextInvisible, stAxisEmpty := PRG_VisuControl.fbVisuControl.arrAxisFrameEmpty[PRG_VisuControl.fbVisuControl.iSelectedAxisPageIndex], stAxis := PRG_VisuControl.fbVisuControl.arrAxisFrame[PRG_VisuControl.fbVisuControl.iSelectedAxisPageIndex], iAxisSelectedPageIndex := PRG_VisuControl.fbVisuControl.iSelectedAxisPageIndex, iAxisTotalPageIndex := PRG_VisuControl.fbVisuControl.iAxisPageIndex)
    Frame (0,199 200x880), frame switch variable: PRG_VisuControl.fbVisuControl.eCurrentNavigation
        shows NavBarEmpty()
        shows NavBarUninitialized(btnInitialize := PRG_VisuControl.fbVisuControl.btnInit)
        shows NavBarInitializing(btnAbort := PRG_VisuControl.fbVisuControl.btnAbort)
        shows NavBarAuto(btnStart := PRG_VisuControl.fbVisuControl.btnStart, btnStop := PRG_VisuControl.fbVisuControl.btnStop, btnManualMode := PRG_VisuControl.fbVisuControl.btnManual, btnAbort := PRG_VisuControl.fbVisuControl.btnAbort, btnReset := PRG_VisuControl.fbVisuControl.btnReset, bVisStart := PRG_VisuControl.fbVisuControl.bStartDisable, bVisStop := PRG_VisuControl.fbVisuControl.bStopDisable)
        shows NavBarManual(btnAutoMode := PRG_VisuControl.fbVisuControl.btnAuto, btnCylinders := PRG_VisuControl.fbVisuControl.btnManualCylinder, btnMotors := PRG_VisuControl.fbVisuControl.btnManualAxis, btnSafety := PRG_VisuControl.fbVisuControl.btnManualSafety, btnInputs := PRG_VisuControl.fbVisuControl.btnManualInputs, btnOutputs := PRG_VisuControl.fbVisuControl.btnManualOutputs, btnOthers := PRG_VisuControl.fbVisuControl.btnManualOthers, btnAbort := PRG_VisuControl.fbVisuControl.btnAbort, btnRobots := PRG_VisuControl.fbVisuControl.btnManualRobots)
        shows NavBarUtilities(btnBack := PRG_VisuControl.fbVisuControl.btnBack)
END_VISUALIZATION

// ---- VISUs/Manual/SingleAxis.TcVIS
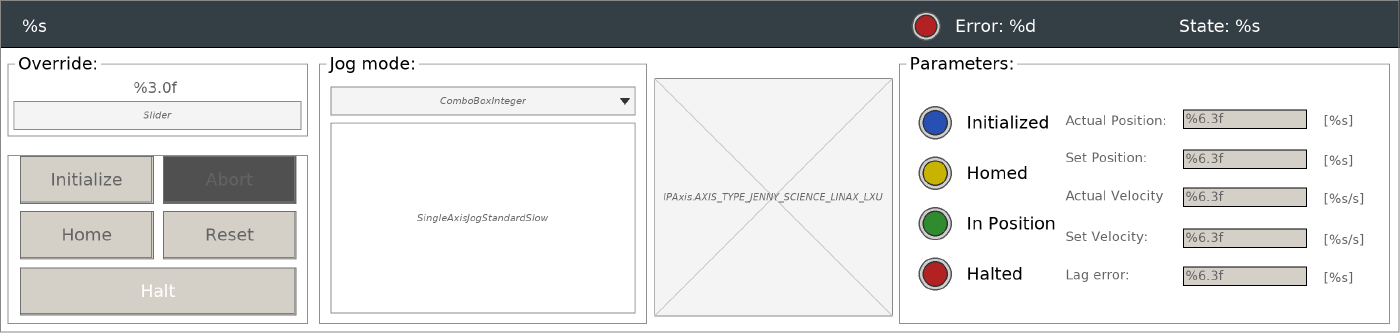
VISUALIZATION SingleAxis  // 1470x350
VAR_IN_OUT
	stAxis : ST_VisuCtrlAxisFrame;
END_VAR
    Rectangle (0,0 1470x50)
    Textfield (20,10 699x35), "%s", text variable: stAxis.sName
    Textfield (1235,10 225x35), "State: %s", text list: 'TL_SingleAxisState', text index: stAxis.eAxisState
    Lamp1 (955,10 35x35), variable: stAxis.bError, style: Lamp-Lamp1-Red
    Textfield (1000,10 200x35), "Error: %d", text variable: stAxis.iErrorID
    Image (687,82 250x250), image: IPAxis.AXIS_TYPE_JENNY_SCIENCE_LINAX_LXU
        p84334746: stAxis.sAxisImage
    GroupBox (8,59 315x84), "Override:"
        Slider (6,47 302x30), variable: stAxis.lrOverride, scale 0..100
        Rectangle (55,18 200x30), "%3.0f", text variable: stAxis.lrOverride
    GroupBox (8,155 315x185)
        Button (13,9 140x50), "Initialize"
            tap stAxis.btnInit
        Button (163,9 140x50), "Abort"
            tap stAxis.btnAbort
        Button (13,67 140x50), "Home"
            tap stAxis.btnHome
        Button (163,67 140x50), "Reset"
            tap stAxis.btnReset
        Button (13,126 290x50), "Halt"
            tap stAxis.btnHalt
    GroupBox (335,59 344x281), "Jog mode:"
        Frame (12,70 320x200), frame switch variable: stAxis.eJogMode
            shows SingleAxisJogStandardSlow(btnJogPositive := stAxis.btnJogPositive, btnJogNegative := stAxis.btnJogNegative)
            shows SingleAxisJogStandardFlast(btnJogPositive := stAxis.btnJogPositive, btnJogNegative := stAxis.btnJogNegative)
            shows SingleAxisJogContinous(btnJogPositive := stAxis.btnJogPositive, btnJogNegative := stAxis.btnJogNegative, lrVelocity := stAxis.lrJogVelocity, lrAcceleration := stAxis.lrJogAcceleration, lrDeceleration := stAxis.lrJogDeceleartion, sUnit := stAxis.sUnit)
            shows SingleAxisJogInching(btnJogPositive := stAxis.btnJogPositive, btnJogNegative := stAxis.btnJogNegative, lrPosition := stAxis.lrJogDistance, lrVelocity := stAxis.lrJogVelocity, lrAcceleration := stAxis.lrJogAcceleration, lrDeceleration := stAxis.lrJogDeceleartion, sUnit := stAxis.sUnit)
            shows SingleAxisJogInchingModulo(btnJogPositive := stAxis.btnJogPositive, btnJogNegative := stAxis.btnJogNegative, lrPosition := stAxis.lrJogDistance, lrVelocity := stAxis.lrJogVelocity, lrAcceleration := stAxis.lrJogAcceleration, lrDeceleration := stAxis.lrJogDeceleartion, sUnit := stAxis.sUnit)
        ComboBoxInteger (12,32 320x30), variable: stAxis.eJogMode, text list: 'TL_SingleAxisJogMode'
            p1601986498: ''
    GroupBox (944,59 515x281), "Parameters:"
        Rectangle (298,56 130x20), "%6.3f", text variable: stAxis.lrActualPosition
        Rectangle (443,59 62x18), "[%s]", text variable: stAxis.sUnit
        Rectangle (172,58 110x20), "Actual Position:"
        Lamp1 (18,156 40x40), variable: stAxis.bInPosition, style: Lamp-Lamp1-Green
        Lamp1 (18,50 40x40), variable: stAxis.bActive, style: Lamp-Lamp1-Blue
        Lamp1 (18,103 40x40), variable: stAxis.bHomed, style: Lamp-Lamp1-Yellow
        Label (68,55 100x30), "Initialized"
        Label (68,108 100x30), "Homed"
        Label (68,161 100x30), "In Position"
        Label (68,214 100x30), "Halted"
        Lamp1 (18,209 40x40), variable: stAxis.bHalted, style: Lamp-Lamp1-Red
        Rectangle (172,97 110x20), "Set Position:"
        Rectangle (298,98 130x20), "%6.3f", text variable: stAxis.lrSetPosition
        Rectangle (443,101 62x18), "[%s]", text variable: stAxis.sUnit
        Rectangle (172,137 110x20), "Actual Velocity"
        Rectangle (298,138 130x20), "%6.3f", text variable: stAxis.lrActualVelocity
        Rectangle (443,141 62x18), "[%s/s]", text variable: stAxis.sUnit
        Rectangle (172,180 110x20), "Set Velocity:"
        Rectangle (298,181 130x20), "%6.3f", text variable: stAxis.lrSetVelocity
        Rectangle (443,184 62x18), "[%s/s]", text variable: stAxis.sUnit
        Rectangle (172,220 110x20), "Lag error:"
        Rectangle (298,221 130x20), "%6.3f", text variable: stAxis.lrLagError
        Rectangle (443,224 62x18), "[%s]", text variable: stAxis.sUnit
END_VISUALIZATION

// ---- VISUs/Manual/SingleDigitalInput.TcVIS
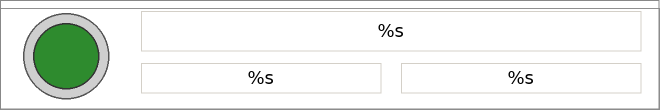
VISUALIZATION SingleDigitalInput  // 660x110
VAR_IN_OUT
	stDigitalInput : ST_VisuCtrlInputFrame;
END_VAR
    GroupBox (0,0 660x110)
        Lamp1 (16,6 100x100), variable: stDigitalInput.bIn, style: Lamp-Lamp1-Green
        Textfield (141,11 500x40), "%s", text variable: stDigitalInput.sName
        Textfield (141,63 240x30), "%s", text variable: stDigitalInput.sModuleType
        Textfield (401,63 240x30), "%s", text variable: stDigitalInput.sPortID
END_VISUALIZATION

// ---- VISUs/Navigation/NavBarAuto.TcVIS
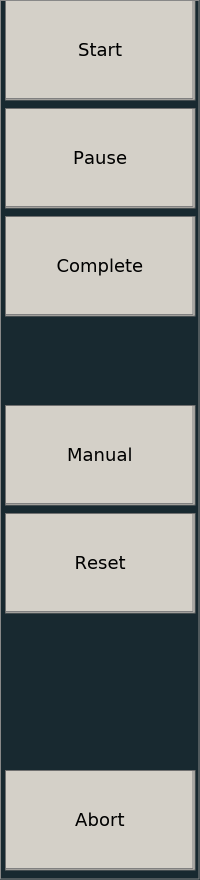
VISUALIZATION NavBarAuto  // 200x880
VAR_IN_OUT
	btnStart 		: BOOL;
	btnStop 		: BOOL;
	btnManualMode	: BOOL;
	btnAbort		: BOOL;
	btnReset		: BOOL;
	
	bVisStart 		: BOOL;
	bVisStop		: BOOL;
END_VAR
    Button (5,0 190x100), "Start", input disabled if: bVisStart
        tap btnStart
    Button (5,108 190x100), "Pause", input disabled if: bVisStop
        tap btnStop
    Button (5,770 190x100), "Abort", input disabled if: bVisStart
        tap btnAbort
    Button (5,405 190x100), "Manual", input disabled if: bVisStart
        tap btnManualMode
    Button (5,513 190x100), "Reset", input disabled if: bVisStart
        tap btnReset
    Button (5,216 190x100), "Complete"
END_VISUALIZATION

// ---- VISUs/Navigation/NavBarAuxilary.TcVIS
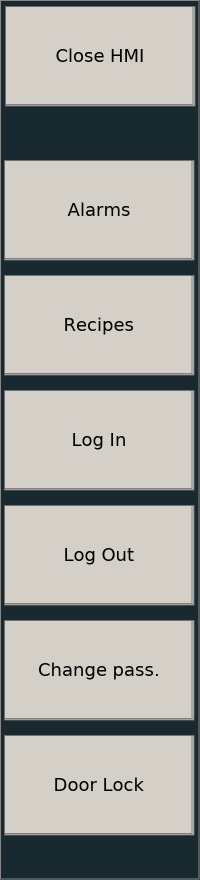
VISUALIZATION NavBarAuxilary  // 200x880
VAR_IN_OUT
	btnAlarms			: BOOL;
	btnRecipes			: BOOL;
	btnDoorLock			: BOOL;
	btnLogIn			: BOOL;
	btnLogOut			: BOOL;
	btnHmiClose			: BOOL;
	sCloseHMIFileName	: STRING;
	sCloseHMIParameters	: STRING;
	
	bVisNotInit 		: BOOL;
	bVisHmiCLose		: BOOL;
	bVisLogIn			: BOOL;
	bVisLogOut			: BOOL;
	bDoorLockDisabled	: BOOL;
	bDoorLockInvisible	: BOOL;
END_VAR
    Button (5,6 190x100), "Close HMI", input disabled if: bVisHmiCLose
        tap btnHmiClose
        toggle btnHmiClose
    Button (4,390 190x100), "Log In", input disabled if: bVisLogIn
        tap btnLogIn
        OnMouseUp: VisuUserMgmt Type=Login
    Button (4,505 190x100), "Log Out", input disabled if: bVisLogOut
        tap btnLogOut
        OnMouseUp: VisuUserMgmt Type=Logout
    Button (4,620 190x100), "Change pass.", input disabled if: bVisLogOut
        OnMouseUp: VisuUserMgmt Type=ChangeUserPassword
    Button (4,160 190x100), "Alarms"
        tap btnAlarms
    Button (4,275 190x100), "Recipes", input disabled if: bVisNotInit
        tap btnRecipes
    Button (4,735 190x100), "Door Lock", invisible if: bDoorLockInvisible, input disabled if: bDoorLockDisabled
        toggle btnDoorLock
END_VISUALIZATION

// ---- VISUs/Navigation/NavBarManual.TcVIS
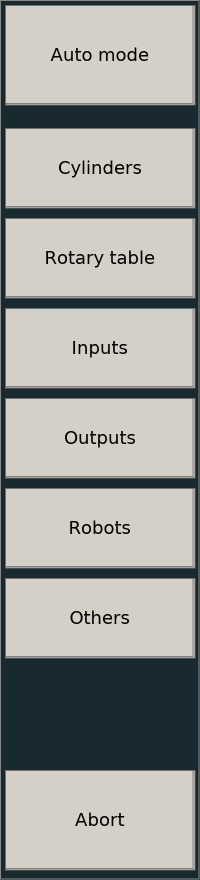
VISUALIZATION NavBarManual  // 200x880
VAR_IN_OUT
	btnAutoMode	: BOOL;
	btnCylinders: BOOL;
	btnMotors	: BOOL;
	btnSafety	: BOOL;
	btnInputs	: BOOL;
	btnOutputs	: BOOL;
	btnOthers	: BOOL;
	btnAbort	: BOOL;
	btnRobots 	: BOOL;
END_VAR
    Button (5,128 190x80), "Cylinders", invisible if: TRUE, input disabled if: TRUE
        tap btnCylinders
    Button (5,218 190x80), "Rotary table"
        tap btnMotors
    Button (5,770 190x100), "Abort"
        tap btnAbort
    Button (5,398 190x80), "Outputs"
        tap btnOutputs
    Button (5,308 190x80), "Inputs"
        tap btnInputs
    Button (5,5 190x100), "Auto mode"
        tap btnAutoMode
    Button (5,578 190x80), "Others"
        tap btnOthers
    Button (5,488 190x80), "Robots"
        tap btnRobots
END_VISUALIZATION

// ---- VISUs/Navigation/NavBarUninitialized.TcVIS
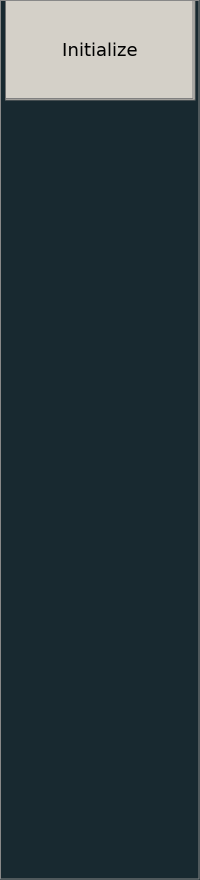
VISUALIZATION NavBarUninitialized  // 200x880
VAR_IN_OUT
	btnInitialize			: BOOL;	(*  *)
END_VAR
    Button (5,0 190x100), "Initialize"
        tap btnInitialize
END_VISUALIZATION

// ---- VISUs/Pages/Auto/AOIBowlFeederFrame.TcVIS
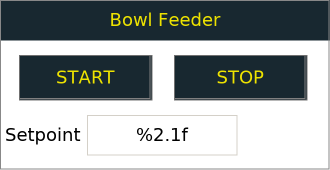
VISUALIZATION AOIBowlFeederFrame  // 330x170
    Rectangle (0,0 330x40), "Bowl Feeder"
    Button (19,55 133x45), "START"
        tap PRG_MachineControl.fbMachineControler.btnStartBowl
    Textfield (87,115 150x40), "%2.1f", text variable: PRG_MachineControl.fbMachineControler.rBowlFeederSetpoint
        OnMouseClick: write the text variable via VisuDialogs.Numpad
    Label (2,120 98x30), "Setpoint"
    Button (174,55 133x45), "STOP"
        tap PRG_MachineControl.fbMachineControler.btnStopBowl
END_VISUALIZATION

// ---- VISUs/Pages/Auto/AOIBatchPerformanceFrame.TcVIS
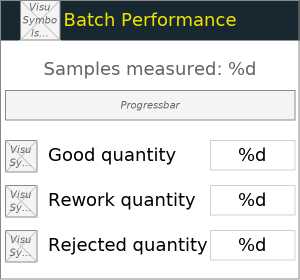
VISUALIZATION AOIBatchPerformanceFrame  // 300x280
VAR_IN_OUT
	stBatchPerformanceFrame : ST_BatchPerformacne;
END_VAR
    Label (45,140 160x30), "Good quantity"
    Label (45,185 160x30), "Rework quantity"
    Label (45,230 160x30), "Rejected quantity"
    Image (5,230 32x32), image: VisuSymbols.Symbols.Wrong
    Image (5,140 32x32), image: VisuSymbols.Symbols.OK
    Image (5,185 32x32), image: VisuSymbols.Symbols.ArrowRoundLeftUp
    Textfield (210,140 85x30), "%d", text variable: stBatchPerformanceFrame.iGoodQuantity
    Textfield (210,185 85x30), "%d", text variable: stBatchPerformanceFrame.iReworkQuantity
    Textfield (210,230 85x30), "%d", text variable: stBatchPerformanceFrame.iRejectedQuantity
    Rectangle (0,0 300x40), "Batch Performance"
    Progressbar (5,90 290x30), variable: stBatchPerformanceFrame.iBatchProgress
    Rectangle (25,54 250x30), "Samples measured: %d", text variable: stBatchPerformanceFrame.iCurrentQuantity
    Image (20,0 40x40), image: VisuSymbols.Symbols.MonitorCurve
END_VISUALIZATION

// ---- VISUs/Pages/Auto/AOIHeaderFrame.TcVIS
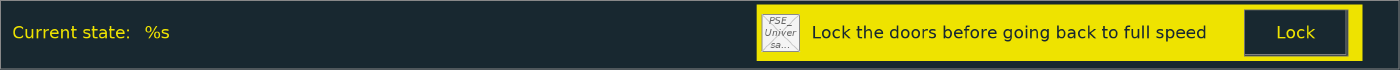
VISUALIZATION AOIHeaderFrame  // 1480x75
VAR_IN_OUT
	eMachineStateAutoFcqText 	: E_MachineCtrlStateAutoFcq;
	stDoorLock	 				: ST_VisuCtrlDoorLock;
END_VAR
    Label (10,15 150x40), "Current state:"
    Textfield (150,15 600x40), "%s", text list: 'TL_Fcq', text index: eMachineStateAutoFcqText
    Frame (800,5 640x60), invisible if: stDoorLock.bDoorLockInvisible
        shows AOIHeaderKeySwitchFrame()
END_VISUALIZATION

// ---- VISUs/Pages/Auto/AOIHeaderKeySwitchFrame.TcVIS
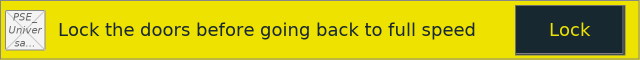
VISUALIZATION AOIHeaderKeySwitchFrame  // 640x60
VAR_IN_OUT
	btnDoorsLock : BOOL;
END_VAR
    Label (55,10 440x40), "Lock the doors before going back to full speed"
    Button (515,5 110x50), "Lock"
        toggle btnDoorsLock
    Image (5,10 40x40), image: PSE_UniversalBlocks.IP_EventSeverity.error
END_VISUALIZATION

// ---- VISUs/Pages/Auto/AOIBatchDataFrame.TcVIS
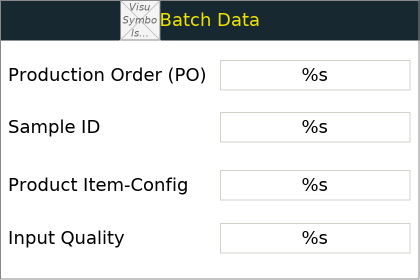
VISUALIZATION AOIBatchDataFrame  // 420x280
VAR_IN_OUT
	stBatchDataFrame : ST_BatchData;
END_VAR
    Label (5,170 210x30), "Product Item-Config"
    Label (5,223 210x30), "Input Quality"
    Textfield (220,170 190x30), "%s", text variable: stBatchDataFrame.sProductItemConfig
    Textfield (220,223 190x30), "%s", text variable: stBatchDataFrame.sInputQuantity
    Rectangle (0,0 420x40), "Batch Data"
    Image (120,0 40x40), image: VisuSymbols.Symbols.Database2
    Label (5,60 210x30), "Production Order (PO)"
    Label (5,112 210x30), "Sample ID"
    Textfield (220,60 190x30), "%s", text variable: stBatchDataFrame.sProductionOrder
    Textfield (220,112 190x30), "%s", text variable: stBatchDataFrame.sTrayID
END_VISUALIZATION

// ---- VISUs/Pages/Auto/AOISortStationFrame.TcVIS
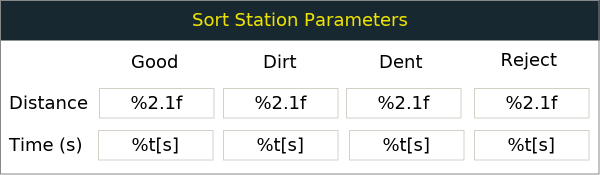
VISUALIZATION AOISortStationFrame  // 600x175
    Rectangle (0,0 600x40), "Sort Station Parameters"
    Label (6,130 90x30), "Time (s)"
    Label (6,88 90x30), "Distance"
    Label (110,47 90x30), "Good"
    Label (235,47 90x30), "Dirt"
    Label (356,47 90x30), "Dent"
    Label (484,45 90x30), "Reject"
    Textfield (99,88 115x30), "%2.1f", text variable: PRG_MachineControl.fbMachineControler.lrSortGoodDistance
        OnMouseClick: write the text variable via VisuDialogs.Numpad
    Textfield (223,88 115x30), "%2.1f", text variable: PRG_MachineControl.fbMachineControler.lrSortDirtDistance
        OnMouseClick: write the text variable via VisuDialogs.Numpad
    Textfield (346,88 115x30), "%2.1f", text variable: PRG_MachineControl.fbMachineControler.lrSortDentDistance
        OnMouseClick: write the text variable via VisuDialogs.Numpad
    Textfield (474,88 115x30), "%2.1f", text variable: PRG_MachineControl.fbMachineControler.lrSortRejectDistance
        OnMouseClick: write the text variable via VisuDialogs.Numpad
    Textfield (98,130 115x30), "%t[s]", text variable: PRG_MachineControl.fbMachineControler.tSortValveGoodTime
        OnMouseClick: write the text variable via VisuDialogs.Numpad
    Textfield (223,130 115x30), "%t[s]", text variable: PRG_MachineControl.fbMachineControler.tSortValveDirtTime
        OnMouseClick: write the text variable via VisuDialogs.Numpad
    Textfield (349,130 115x30), "%t[s]", text variable: PRG_MachineControl.fbMachineControler.tSortValveDentTime
        OnMouseClick: write the text variable via VisuDialogs.Numpad
    Textfield (474,130 115x30), "%t[s]", text variable: PRG_MachineControl.fbMachineControler.tSortValveRejectTime
        OnMouseClick: write the text variable via VisuDialogs.Numpad
END_VISUALIZATION

// ---- VISUs/Pages/Auto/PageAuto.TcVIS
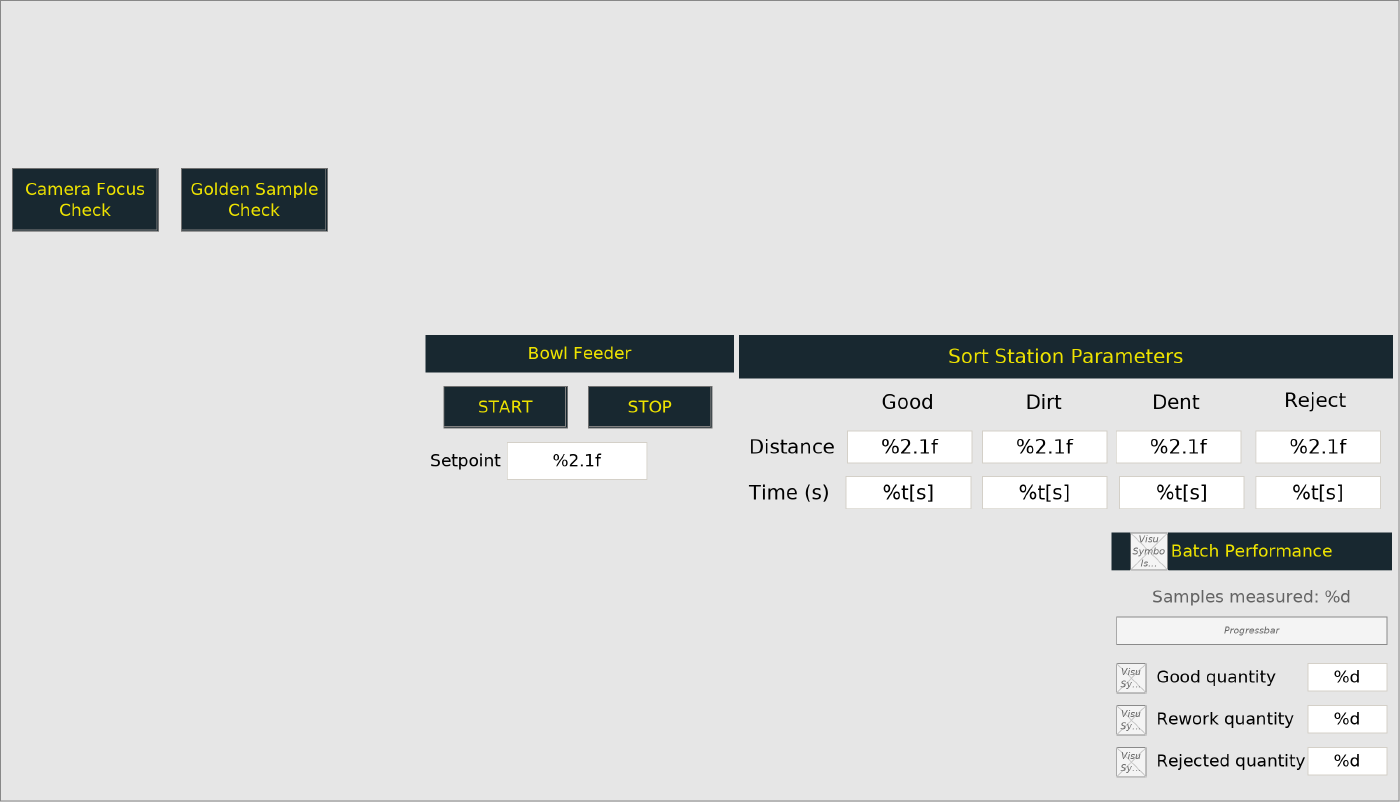
VISUALIZATION PageAuto  // 1500x860
    Frame (792,359 700x204)
        shows AOISortStationFrame()
    Button (13,180 157x68), "Camera Focus Check"
    Button (194,180 157x68), "Golden Sample Check"
    Frame (456,359 330x170)
        shows AOIBowlFeederFrame()
    Frame (1191,571 300x280)
        shows AOIBatchPerformanceFrame(stBatchPerformanceFrame := PRG_MachineControl.fbMachineControler.stBatchPerformance)
END_VISUALIZATION

// ---- VISUs/Pages/Initializing/InitializingDoorLockOpen.TcVIS
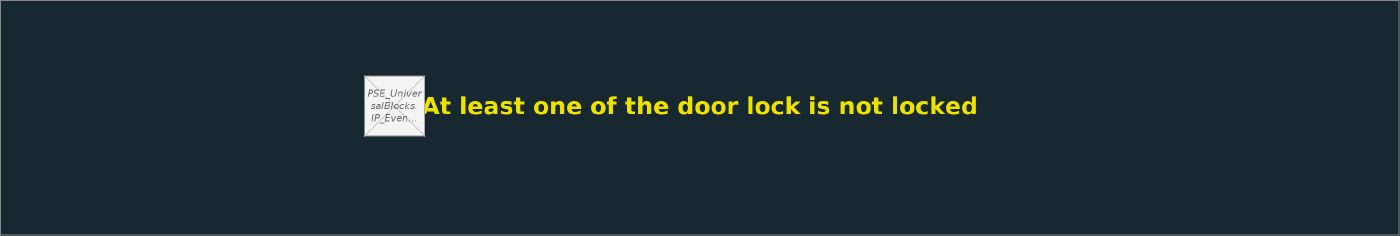
VISUALIZATION InitializingDoorLockOpen  // 1480x250
    Label (0,92 1480x40), "At least one of the door lock is not locked"
    Image (385,80 64x64), image: PSE_UniversalBlocks.IP_EventSeverity.error
END_VISUALIZATION

// ---- VISUs/Pages/Initializing/InitializingEStopActive.TcVIS
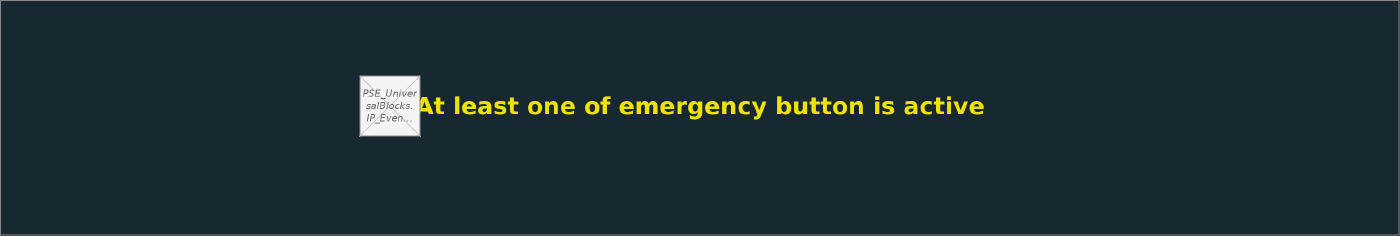
VISUALIZATION InitializingEStopActive  // 1480x250
    Label (0,92 1480x40), "At least one of emergency button is active"
    Image (380,80 64x64), image: PSE_UniversalBlocks.IP_EventSeverity.error
END_VISUALIZATION

// ---- VISUs/Pages/Initializing/InitializingFixtureConnectionFailed.TcVIS
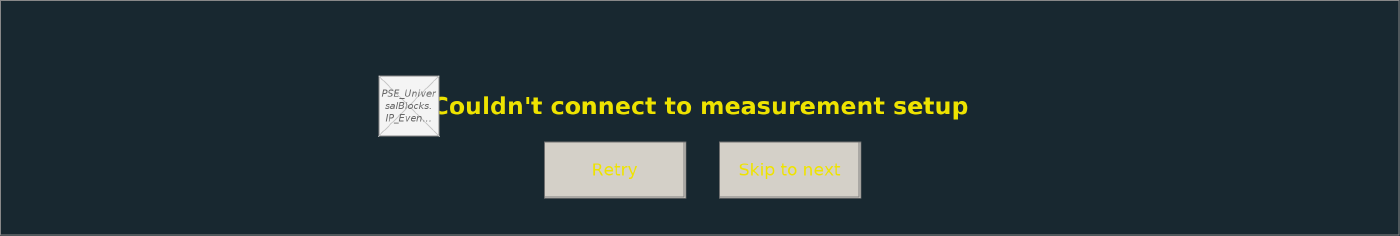
VISUALIZATION InitializingFixtureConnectionFailed  // 1480x250
VAR_IN_OUT
	btnFixtureConnectionRetry	: BOOL;
	btnFixtureConnectionSkip	: BOOL;
END_VAR
    Label (0,92 1480x40), "Couldn't connect to measurement setup"
    Button (575,150 150x60), "Retry"
        toggle btnFixtureConnectionRetry
    Button (760,150 150x60), "Skip to next"
        toggle btnFixtureConnectionSkip
    Image (400,80 64x64), image: PSE_UniversalBlocks.IP_EventSeverity.warning
END_VISUALIZATION

// ---- VISUs/Pages/Initializing/InitializingNoFixturesAvailable.TcVIS
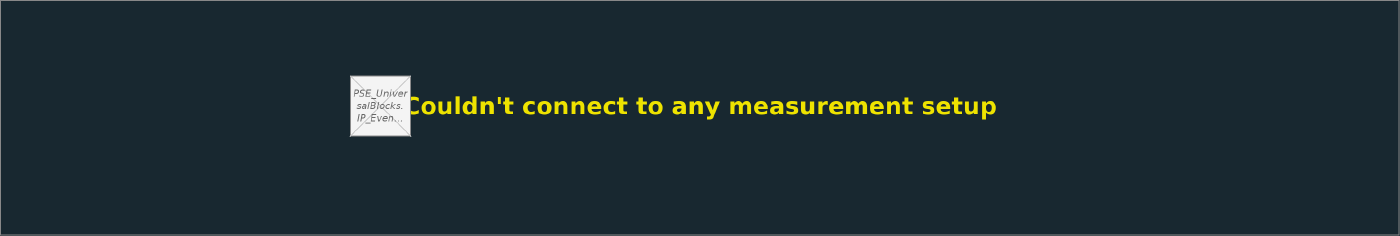
VISUALIZATION InitializingNoFixturesAvailable  // 1480x250
    Label (0,92 1480x40), "Couldn't connect to any measurement setup"
    Image (370,80 64x64), image: PSE_UniversalBlocks.IP_EventSeverity.critical
END_VISUALIZATION

// ---- VISUs/Pages/Initializing/InitializingRotaryTablePlaceTrayDialog.TcVIS
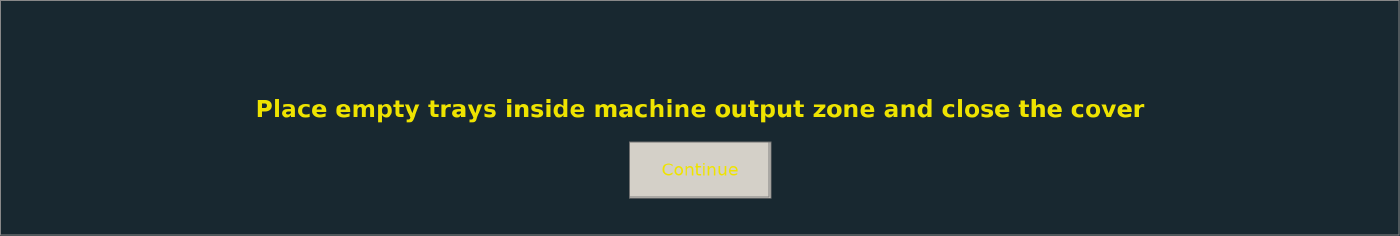
VISUALIZATION InitializingRotaryTablePlaceTrayDialog  // 1480x250
VAR_IN_OUT
	stInitializationRotaryTableFrame : ST_InitializationRotaryTableFrame;
END_VAR
    Label (0,95 1480x40), "Place empty trays inside machine output zone and close the cover"
    Button (665,150 150x60), "Continue", input disabled if: stInitializationRotaryTableFrame.bContinueDisabled
        toggle stInitializationRotaryTableFrame.btnContinue
END_VISUALIZATION

// ---- VISUs/Pages/Initializing/InitializingStartSafetySystem.TcVIS
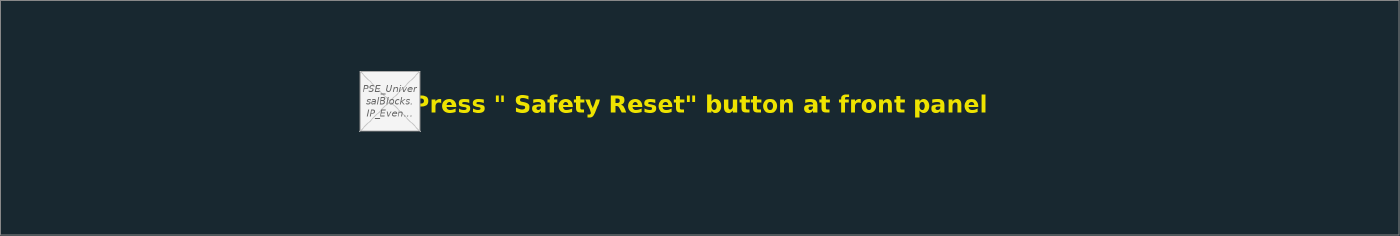
VISUALIZATION InitializingStartSafetySystem  // 1480x250
    Label (0,95 1480x30), "Press " Safety Reset" button at front panel"
    Image (380,75 64x64), image: PSE_UniversalBlocks.IP_EventSeverity.info
END_VISUALIZATION

// ---- VISUs/Pages/Initializing/InitializingTrayfeederCourtainBroken.TcVIS
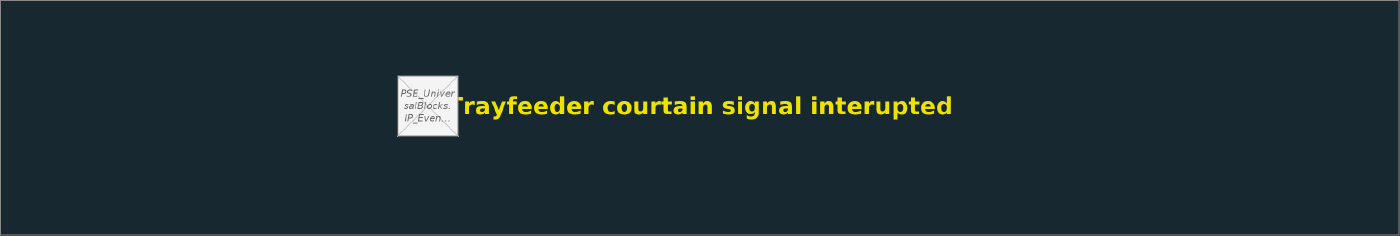
VISUALIZATION InitializingTrayfeederCourtainBroken  // 1480x250
    Label (0,92 1480x40), "Trayfeeder courtain signal interupted"
    Image (420,80 64x64), image: PSE_UniversalBlocks.IP_EventSeverity.error
END_VISUALIZATION

